// TIA Portal project "application-cp" (V18)

(* hardware
DEVICE "S7-1200 station_1"  S7-1200 Station
   slot 0: "Rack_0"  S7-1200 Rack  Rack  V1.0
   slot 1: "cpu"  CPU 1215C DC/DC/DC  6ES7 215-1AG40-0XB0  V4.6
*)

// ===== PLC "cpu"  CPU 1215C DC/DC/DC =====

VAR_GLOBAL   // PLC tag table "Default tag table"
   "Clock_Byte" AT %MB0 : Byte;
   "Clock_10Hz" AT %M0.0 : Bool;
   "Clock_5Hz" AT %M0.1 : Bool;
   "Clock_2.5Hz" AT %M0.2 : Bool;
   "Clock_2Hz" AT %M0.3 : Bool;
   "Clock_1.25Hz" AT %M0.4 : Bool;
   "Clock_1Hz" AT %M0.5 : Bool;
   "Clock_0.625Hz" AT %M0.6 : Bool;
   "Clock_0.5Hz" AT %M0.7 : Bool;
   "System_Byte" AT %MB1 : Byte;
   "FirstScan" AT %M1.0 : Bool;
   "DiagStatusUpdate" AT %M1.1 : Bool;
   "AlwaysTRUE" AT %M1.2 : Bool;
   "AlwaysFALSE" AT %M1.3 : Bool;
   "Tag_1" AT %M10.0 : Bool;
   "Tag_2" AT %M30.0 : Bool;
   "Tag_3" AT %M30.1 : Bool;
   "Tag_4" AT %M30.2 : Bool;
   "Tag_5" AT %M30.3 : Bool;
   "Tag_6" AT %M30.4 : Bool;
   "Tag_7" AT %M30.5 : Bool;
   "Tag_8" AT %M30.6 : Bool;
   "Tag_9" AT %M30.7 : Bool;
   "Tag_10" AT %M31.0 : Bool;
   "Tag_11" AT %M31.2 : Bool;
   "Tag_12" AT %M31.1 : Bool;
   "Tag_13" AT %M31.3 : Bool;
   "Tag_14" AT %M40.0 : Bool;
   "Tag_15" AT %M40.1 : Bool;
   "Tag_16" AT %M40.2 : Bool;
   "Tag_17" AT %M40.3 : Bool;
   "Tag_18" AT %M40.4 : Bool;
   "Tag_19" AT %M40.5 : Bool;
   "Tag_20" AT %M40.6 : Bool;
   "Tag_21" AT %M40.7 : Bool;
   "Tag_22" AT %M41.0 : Bool;
   "Tag_23" AT %M41.1 : Bool;
   "Tag_24" AT %M41.2 : Bool;
   "Tag_25" AT %M41.3 : Bool;
   "Tag_26" AT %M41.4 : Bool;
   "Tag_27" AT %M31.4 : Bool;
   "Tag_28" AT %M31.5 : Bool;
   "Tag_29" AT %M41.5 : Bool;
   "Tag_30" AT %M41.6 : Bool;
   "Tag_31" AT %M41.7 : Bool;
   "Tag_32" AT %M42.0 : Bool;
   "Tag_33" AT %M31.6 : Bool;
   "Tag_34" AT %M42.1 : Bool;
   "Tag_35" AT %M50.0 : Bool;
   "Tag_36" AT %M60.0 : Bool;
   "Tag_37" AT %M60.1 : Bool;
   "Tag_38" AT %M70.0 : Bool;
   "Tag_39" AT %M70.1 : Bool;
   "Tag_40" AT %M70.2 : Bool;
   "Tag_41" AT %M70.3 : Bool;
   "Tag_42" AT %M80.0 : Bool;
   "Tag_43" AT %M80.1 : Bool;
   "Tag_44" AT %M90.0 : Bool;
   "Tag_45" AT %M90.1 : Bool;
   "Tag_46" AT %M100.0 : Bool;
   "Tag_47" AT %M100.1 : Bool;
   "Tag_48" AT %M11.0 : Bool;
   "Tag_49" AT %M110.0 : Bool;
   "Tag_50" AT %M110.1 : Bool;
   "Tag_51" AT %M120.0 : Bool;
   "Tag_52" AT %M120.1 : Bool;
   "Tag_53" AT %M50.1 : Bool;
   "Tag_54" AT %M50.2 : Bool;
   "Tag_55" AT %M50.3 : Bool;
   "Tag_56" AT %M50.4 : Bool;
   "Tag_57" AT %M50.5 : Bool;
   "Tag_58" AT %M50.6 : Bool;
   "Tag_59" AT %M50.7 : Bool;
END_VAR

TYPE "Tank"
   STRUCT
      ID : Int;
      Sensor : Struct
         High : Bool;
         Low : Bool := true;
      END_STRUCT;
      Valve : Struct
         Drain : Bool;
         Source : Bool;
      END_STRUCT;
      Object : Struct
         Motor : Bool;
         Pump : Bool;
      END_STRUCT;
   END_STRUCT;
END_TYPE

TYPE "Line"
   STRUCT
      Supply : Struct
         Pump : Bool;
         Valve : Struct
            Caustic : Bool;
            Acid : Bool;
            Water : Bool;
            Rinse : Bool;
            Rice : Bool;
            Malt : Bool;
            Filter : Bool;
            Hops : Bool;
            Settling : Bool;
         END_STRUCT;
      END_STRUCT;
      "Return" : Struct
         Pump : Bool;
         Valve : Struct
            Caustic : Bool;
            Acid : Bool;
            Water : Bool;
            Rinse : Bool;
            Drain : Bool;
         END_STRUCT;
      END_STRUCT;
   END_STRUCT;
END_TYPE

DATA_BLOCK "DB_Tagforce"   // DB1
{ S7_Optimized_Access := 'FALSE' }
VERSION : 0.1
   VAR
      Button : Struct
         Run : Bool;
         Start : Bool;
         Mode : Bool;
         Clean : Struct
            Rice : Bool;
            Malt : Bool;
            Filter : Bool;
            Hops : Bool;
            Settling : Bool;
         END_STRUCT;
      END_STRUCT;
      Status : Struct
         Program : Struct
            Online : Bool;
            Offline : Bool;
            Idle : Bool;
            Busy : Bool;
         END_STRUCT;
         Mode : Struct
            Manual : Bool;
            Automatic : Bool;
         END_STRUCT;
         "Step" : Struct
            "1" : Bool;
            "2" : Bool;
            "3" : Bool;
            "4" : Bool;
            "5" : Bool;
            "6" : Bool;
            "7" : Bool;
         END_STRUCT;
         Clean : Struct
            Rice : Bool;
            Malt : Bool;
            Filter : Bool;
            Hops : Bool;
            Settling : Bool;
         END_STRUCT;
         Done : Bool;
      END_STRUCT;
      Lock : Struct
         Mode : Bool;
         "Step" : Struct
            "1" : Bool;
            "2" : Bool;
            "3" : Bool;
            "4" : Bool;
            "5" : Bool;
            "6" : Bool;
            "7" : Bool;
         END_STRUCT;
         Clean : Bool;
      END_STRUCT;
   END_VAR
BEGIN
END_DATA_BLOCK

DATA_BLOCK "DB_Tanks"   // DB2
{ S7_Optimized_Access := 'FALSE' }
VERSION : 0.1
   VAR
      Source : Struct
         Caustic : "Tank";
         Acid : "Tank";
         Water : "Tank";
         Rinse : "Tank";
      END_STRUCT;
      CIP : Struct
         Rice : "Tank";
         Malt : "Tank";
         Filter : "Tank";
         Hops : "Tank";
         Settling : "Tank";
         Current : "Tank";
         Backup : "Tank";
      END_STRUCT;
   END_VAR
BEGIN
   Source.Caustic.ID := 1;
   Source.Acid.ID := 2;
   Source.Water.ID := 3;
   Source.Rinse.ID := 4;
   CIP.Rice.ID := 5;
   CIP.Malt.ID := 6;
   CIP.Filter.ID := 7;
   CIP.Hops.ID := 8;
   CIP.Settling.ID := 9;
END_DATA_BLOCK

DATA_BLOCK "DB_Lines"   // DB3
{ S7_Optimized_Access := 'FALSE' }
VERSION : 0.1
   VAR
      Line : "Line";
   END_VAR
BEGIN
END_DATA_BLOCK

DATA_BLOCK "DB_Counter"   // DB37
{ S7_Optimized_Access := 'FALSE' }
VERSION : 0.1
   VAR
      Rice : Bool;
      Malt : Bool;
      Filter : Bool;
      Hops : Bool;
      Settling : Bool;
      Caustic : Bool;
      Acid : Bool;
      Water : Bool;
      Rinse : Bool;
      S7 : Bool;
      CC : Bool;
      CA : Bool;
      LM : Bool;
   END_VAR
BEGIN
END_DATA_BLOCK

// folder: System blocks/Program resources

DATA_BLOCK "IEC_Timer_0_DB"   // DB4
{ S7_Optimized_Access := 'TRUE' }
AUTHOR : Simatic
FAMILY : IEC
NAME : IEC_TMR
VERSION : 1.0
// stored: InstanceOfName IEC_TIMER
"IEC_TIMER"
BEGIN
END_DATA_BLOCK

DATA_BLOCK "IEC_Timer_0_DB_1"   // DB5
{ S7_Optimized_Access := 'TRUE' }
AUTHOR : Simatic
FAMILY : IEC
NAME : IEC_TMR
VERSION : 1.0
// stored: InstanceOfName IEC_TIMER
"IEC_TIMER"
BEGIN
END_DATA_BLOCK

DATA_BLOCK "IEC_Timer_0_DB_2"   // DB6
{ S7_Optimized_Access := 'TRUE' }
AUTHOR : Simatic
FAMILY : IEC
NAME : IEC_TMR
VERSION : 1.0
// stored: InstanceOfName IEC_TIMER
"IEC_TIMER"
BEGIN
END_DATA_BLOCK

DATA_BLOCK "IEC_Timer_0_DB_3"   // DB7
{ S7_Optimized_Access := 'TRUE' }
AUTHOR : Simatic
FAMILY : IEC
NAME : IEC_TMR
VERSION : 1.0
// stored: InstanceOfName IEC_TIMER
"IEC_TIMER"
BEGIN
END_DATA_BLOCK

DATA_BLOCK "IEC_Timer_0_DB_4"   // DB8
{ S7_Optimized_Access := 'TRUE' }
AUTHOR : Simatic
FAMILY : IEC
NAME : IEC_TMR
VERSION : 1.0
// stored: InstanceOfName IEC_TIMER
"IEC_TIMER"
BEGIN
END_DATA_BLOCK

DATA_BLOCK "IEC_Timer_0_DB_5"   // DB9
{ S7_Optimized_Access := 'TRUE' }
AUTHOR : Simatic
FAMILY : IEC
NAME : IEC_TMR
VERSION : 1.0
// stored: InstanceOfName IEC_TIMER
"IEC_TIMER"
BEGIN
END_DATA_BLOCK

DATA_BLOCK "IEC_Timer_0_DB_6"   // DB10
{ S7_Optimized_Access := 'TRUE' }
AUTHOR : Simatic
FAMILY : IEC
NAME : IEC_TMR
VERSION : 1.0
// stored: InstanceOfName IEC_TIMER
"IEC_TIMER"
BEGIN
END_DATA_BLOCK

DATA_BLOCK "IEC_Timer_0_DB_7"   // DB11
{ S7_Optimized_Access := 'TRUE' }
AUTHOR : Simatic
FAMILY : IEC
NAME : IEC_TMR
VERSION : 1.0
// stored: InstanceOfName IEC_TIMER
"IEC_TIMER"
BEGIN
END_DATA_BLOCK

DATA_BLOCK "IEC_Timer_0_DB_8"   // DB12
{ S7_Optimized_Access := 'TRUE' }
AUTHOR : Simatic
FAMILY : IEC
NAME : IEC_TMR
VERSION : 1.0
// stored: InstanceOfName IEC_TIMER
"IEC_TIMER"
BEGIN
END_DATA_BLOCK

DATA_BLOCK "IEC_Timer_0_DB_9"   // DB13
{ S7_Optimized_Access := 'TRUE' }
AUTHOR : Simatic
FAMILY : IEC
NAME : IEC_TMR
VERSION : 1.0
// stored: InstanceOfName IEC_TIMER
"IEC_TIMER"
BEGIN
END_DATA_BLOCK

DATA_BLOCK "IEC_Timer_0_DB_10"   // DB14
{ S7_Optimized_Access := 'TRUE' }
AUTHOR : Simatic
FAMILY : IEC
NAME : IEC_TMR
VERSION : 1.0
// stored: InstanceOfName IEC_TIMER
"IEC_TIMER"
BEGIN
END_DATA_BLOCK

DATA_BLOCK "IEC_Timer_0_DB_11"   // DB15
{ S7_Optimized_Access := 'TRUE' }
AUTHOR : Simatic
FAMILY : IEC
NAME : IEC_TMR
VERSION : 1.0
// stored: InstanceOfName IEC_TIMER
"IEC_TIMER"
BEGIN
END_DATA_BLOCK

DATA_BLOCK "IEC_Timer_0_DB_12"   // DB16
{ S7_Optimized_Access := 'TRUE' }
AUTHOR : Simatic
FAMILY : IEC
NAME : IEC_TMR
VERSION : 1.0
// stored: InstanceOfName IEC_TIMER
"IEC_TIMER"
BEGIN
END_DATA_BLOCK

DATA_BLOCK "IEC_Timer_0_DB_13"   // DB17
{ S7_Optimized_Access := 'TRUE' }
AUTHOR : Simatic
FAMILY : IEC
NAME : IEC_TMR
VERSION : 1.0
// stored: InstanceOfName IEC_TIMER
"IEC_TIMER"
BEGIN
END_DATA_BLOCK

DATA_BLOCK "IEC_Timer_0_DB_14"   // DB18
{ S7_Optimized_Access := 'TRUE' }
AUTHOR : Simatic
FAMILY : IEC
NAME : IEC_TMR
VERSION : 1.0
// stored: InstanceOfName IEC_TIMER
"IEC_TIMER"
BEGIN
END_DATA_BLOCK

DATA_BLOCK "IEC_Timer_0_DB_15"   // DB19
{ S7_Optimized_Access := 'TRUE' }
AUTHOR : Simatic
FAMILY : IEC
NAME : IEC_TMR
VERSION : 1.0
// stored: InstanceOfName IEC_TIMER
"IEC_TIMER"
BEGIN
END_DATA_BLOCK

DATA_BLOCK "IEC_Timer_0_DB_16"   // DB20
{ S7_Optimized_Access := 'TRUE' }
AUTHOR : Simatic
FAMILY : IEC
NAME : IEC_TMR
VERSION : 1.0
// stored: InstanceOfName IEC_TIMER
"IEC_TIMER"
BEGIN
END_DATA_BLOCK

DATA_BLOCK "IEC_Timer_0_DB_17"   // DB21
{ S7_Optimized_Access := 'TRUE' }
AUTHOR : Simatic
FAMILY : IEC
NAME : IEC_TMR
VERSION : 1.0
// stored: InstanceOfName IEC_TIMER
"IEC_TIMER"
BEGIN
END_DATA_BLOCK

DATA_BLOCK "IEC_Timer_0_DB_18"   // DB22
{ S7_Optimized_Access := 'TRUE' }
AUTHOR : Simatic
FAMILY : IEC
NAME : IEC_TMR
VERSION : 1.0
// stored: InstanceOfName IEC_TIMER
"IEC_TIMER"
BEGIN
END_DATA_BLOCK

DATA_BLOCK "IEC_Timer_0_DB_19"   // DB23
{ S7_Optimized_Access := 'TRUE' }
AUTHOR : Simatic
FAMILY : IEC
NAME : IEC_TMR
VERSION : 1.0
// stored: InstanceOfName IEC_TIMER
"IEC_TIMER"
BEGIN
END_DATA_BLOCK

DATA_BLOCK "IEC_Timer_0_DB_20"   // DB24
{ S7_Optimized_Access := 'TRUE' }
AUTHOR : Simatic
FAMILY : IEC
NAME : IEC_TMR
VERSION : 1.0
// stored: InstanceOfName IEC_TIMER
"IEC_TIMER"
BEGIN
END_DATA_BLOCK

DATA_BLOCK "IEC_Timer_0_DB_21"   // DB25
{ S7_Optimized_Access := 'TRUE' }
AUTHOR : Simatic
FAMILY : IEC
NAME : IEC_TMR
VERSION : 1.0
// stored: InstanceOfName IEC_TIMER
"IEC_TIMER"
BEGIN
END_DATA_BLOCK

DATA_BLOCK "IEC_Timer_0_DB_22"   // DB26
{ S7_Optimized_Access := 'TRUE' }
AUTHOR : Simatic
FAMILY : IEC
NAME : IEC_TMR
VERSION : 1.0
// stored: InstanceOfName IEC_TIMER
"IEC_TIMER"
BEGIN
END_DATA_BLOCK

DATA_BLOCK "IEC_Timer_0_DB_23"   // DB27
{ S7_Optimized_Access := 'TRUE' }
AUTHOR : Simatic
FAMILY : IEC
NAME : IEC_TMR
VERSION : 1.0
// stored: InstanceOfName IEC_TIMER
"IEC_TIMER"
BEGIN
END_DATA_BLOCK

DATA_BLOCK "IEC_Timer_0_DB_24"   // DB28
{ S7_Optimized_Access := 'TRUE' }
AUTHOR : Simatic
FAMILY : IEC
NAME : IEC_TMR
VERSION : 1.0
// stored: InstanceOfName IEC_TIMER
"IEC_TIMER"
BEGIN
END_DATA_BLOCK

DATA_BLOCK "IEC_Timer_0_DB_25"   // DB29
{ S7_Optimized_Access := 'TRUE' }
AUTHOR : Simatic
FAMILY : IEC
NAME : IEC_TMR
VERSION : 1.0
// stored: InstanceOfName IEC_TIMER
"IEC_TIMER"
BEGIN
END_DATA_BLOCK

DATA_BLOCK "IEC_Timer_0_DB_26"   // DB30
{ S7_Optimized_Access := 'TRUE' }
AUTHOR : Simatic
FAMILY : IEC
NAME : IEC_TMR
VERSION : 1.0
// stored: InstanceOfName IEC_TIMER
"IEC_TIMER"
BEGIN
END_DATA_BLOCK

DATA_BLOCK "IEC_Timer_0_DB_27"   // DB31
{ S7_Optimized_Access := 'TRUE' }
AUTHOR : Simatic
FAMILY : IEC
NAME : IEC_TMR
VERSION : 1.0
// stored: InstanceOfName IEC_TIMER
"IEC_TIMER"
BEGIN
END_DATA_BLOCK

DATA_BLOCK "IEC_Timer_0_DB_28"   // DB32
{ S7_Optimized_Access := 'TRUE' }
AUTHOR : Simatic
FAMILY : IEC
NAME : IEC_TMR
VERSION : 1.0
// stored: InstanceOfName IEC_TIMER
"IEC_TIMER"
BEGIN
END_DATA_BLOCK

DATA_BLOCK "IEC_Timer_0_DB_29"   // DB33
{ S7_Optimized_Access := 'TRUE' }
AUTHOR : Simatic
FAMILY : IEC
NAME : IEC_TMR
VERSION : 1.0
// stored: InstanceOfName IEC_TIMER
"IEC_TIMER"
BEGIN
END_DATA_BLOCK

DATA_BLOCK "IEC_Timer_0_DB_30"   // DB34
{ S7_Optimized_Access := 'TRUE' }
AUTHOR : Simatic
FAMILY : IEC
NAME : IEC_TMR
VERSION : 1.0
// stored: InstanceOfName IEC_TIMER
"IEC_TIMER"
BEGIN
END_DATA_BLOCK

// folder: (top level)

ORGANIZATION_BLOCK "Main"   // OB1, LAD, ProgramCycle
TITLE = "Main Program Sweep (Cycle)"
{ S7_Optimized_Access := 'TRUE' }
VERSION : 0.1
   VAR_INPUT
      Initial_Call : Bool;   // Initial call of this OB
      Remanence : Bool;   // =True, if remanent data are available
   END_VAR
   VAR_TEMP   // added for the SCL form of the ladder/FBD networks
      _w1 : Bool;
      _w2 : Bool;
      _w3 : Bool;
      _w4 : Bool;
      _w5 : Bool;
      _w6 : Bool;
      _w7 : Bool;
      _w8 : Bool;
      _w9 : Bool;
      _w10 : Bool;
      _w11 : Bool;
      _w12 : Bool;
      _w13 : Bool;
      _w14 : Bool;
      _w15 : Bool;
      _w16 : Bool;
   END_VAR
BEGIN

REGION Network 1: Program
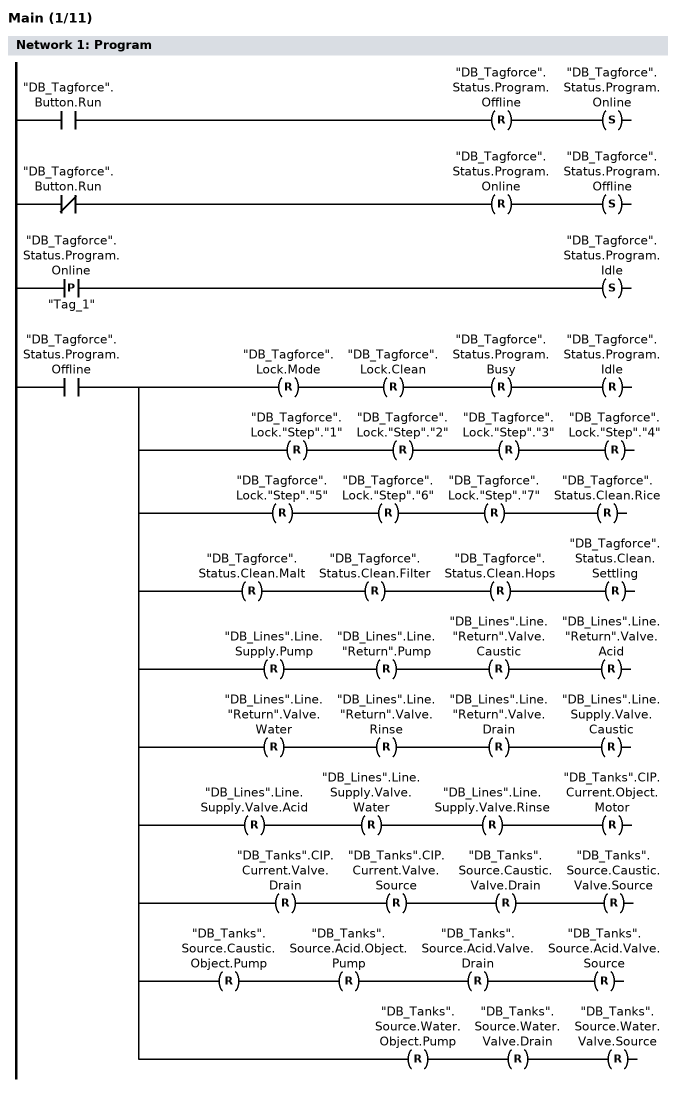
   RUNG wire#powerrail
      Contact( "DB_Tagforce".Button.Run )
      R_Coil( "DB_Tagforce".Status.Program.Offline )
      S_Coil( "DB_Tagforce".Status.Program.Online )
   END_RUNG
   RUNG wire#powerrail
      I_Contact( "DB_Tagforce".Button.Run )
      R_Coil( "DB_Tagforce".Status.Program.Online )
      S_Coil( "DB_Tagforce".Status.Program.Offline )
   END_RUNG
   RUNG wire#powerrail
      P_Contact(operand := "DB_Tagforce".Status.Program.Online, bit := "Tag_1")
      S_Coil( "DB_Tagforce".Status.Program.Idle )
   END_RUNG
   RUNG wire#powerrail
      Contact( "DB_Tagforce".Status.Program.Offline )
      wire#w1
      R_Coil( "DB_Tagforce".Lock.Mode )
      R_Coil( "DB_Tagforce".Lock.Clean )
      R_Coil( "DB_Tagforce".Status.Program.Busy )
      R_Coil( "DB_Tagforce".Status.Program.Idle )
   END_RUNG
   RUNG wire#w1
      R_Coil( "DB_Tagforce".Lock."Step"."1" )
      R_Coil( "DB_Tagforce".Lock."Step"."2" )
      R_Coil( "DB_Tagforce".Lock."Step"."3" )
      R_Coil( "DB_Tagforce".Lock."Step"."4" )
   END_RUNG
   RUNG wire#w1
      R_Coil( "DB_Tagforce".Lock."Step"."5" )
      R_Coil( "DB_Tagforce".Lock."Step"."6" )
      R_Coil( "DB_Tagforce".Lock."Step"."7" )
      R_Coil( "DB_Tagforce".Status.Clean.Rice )
   END_RUNG
   RUNG wire#w1
      R_Coil( "DB_Tagforce".Status.Clean.Malt )
      R_Coil( "DB_Tagforce".Status.Clean.Filter )
      R_Coil( "DB_Tagforce".Status.Clean.Hops )
      R_Coil( "DB_Tagforce".Status.Clean.Settling )
   END_RUNG
   RUNG wire#w1
      R_Coil( "DB_Lines".Line.Supply.Pump )
      R_Coil( "DB_Lines".Line."Return".Pump )
      R_Coil( "DB_Lines".Line."Return".Valve.Caustic )
      R_Coil( "DB_Lines".Line."Return".Valve.Acid )
   END_RUNG
   RUNG wire#w1
      R_Coil( "DB_Lines".Line."Return".Valve.Water )
      R_Coil( "DB_Lines".Line."Return".Valve.Rinse )
      R_Coil( "DB_Lines".Line."Return".Valve.Drain )
      R_Coil( "DB_Lines".Line.Supply.Valve.Caustic )
   END_RUNG
   RUNG wire#w1
      R_Coil( "DB_Lines".Line.Supply.Valve.Acid )
      R_Coil( "DB_Lines".Line.Supply.Valve.Water )
      R_Coil( "DB_Lines".Line.Supply.Valve.Rinse )
      R_Coil( "DB_Tanks".CIP.Current.Object.Motor )
   END_RUNG
   RUNG wire#w1
      R_Coil( "DB_Tanks".CIP.Current.Valve.Drain )
      R_Coil( "DB_Tanks".CIP.Current.Valve.Source )
      R_Coil( "DB_Tanks".Source.Caustic.Valve.Drain )
      R_Coil( "DB_Tanks".Source.Caustic.Valve.Source )
   END_RUNG
   RUNG wire#w1
      R_Coil( "DB_Tanks".Source.Caustic.Object.Pump )
      R_Coil( "DB_Tanks".Source.Acid.Object.Pump )
      R_Coil( "DB_Tanks".Source.Acid.Valve.Drain )
      R_Coil( "DB_Tanks".Source.Acid.Valve.Source )
   END_RUNG
   RUNG wire#w1
      R_Coil( "DB_Tanks".Source.Water.Object.Pump )
      R_Coil( "DB_Tanks".Source.Water.Valve.Drain )
      R_Coil( "DB_Tanks".Source.Water.Valve.Source )
   END_RUNG
   // the same network as SCL:
   IF "DB_Tagforce".Button.Run THEN
       "DB_Tagforce".Status.Program.Offline := FALSE;
       "DB_Tagforce".Status.Program.Online := TRUE;
   END_IF;
   IF NOT "DB_Tagforce".Button.Run THEN
       "DB_Tagforce".Status.Program.Online := FALSE;
       "DB_Tagforce".Status.Program.Offline := TRUE;
   END_IF;
   #_w1 := "DB_Tagforce".Status.Program.Online AND NOT "Tag_1";   // rising edge of "DB_Tagforce".Status.Program.Online
   "Tag_1" := "DB_Tagforce".Status.Program.Online;
   IF #_w1 THEN "DB_Tagforce".Status.Program.Idle := TRUE; END_IF;
   IF "DB_Tagforce".Status.Program.Offline THEN
       "DB_Tagforce".Lock.Mode := FALSE;
       "DB_Tagforce".Lock.Clean := FALSE;
       "DB_Tagforce".Status.Program.Busy := FALSE;
       "DB_Tagforce".Status.Program.Idle := FALSE;
       "DB_Tagforce".Lock."Step"."1" := FALSE;
       "DB_Tagforce".Lock."Step"."2" := FALSE;
       "DB_Tagforce".Lock."Step"."3" := FALSE;
       "DB_Tagforce".Lock."Step"."4" := FALSE;
       "DB_Tagforce".Lock."Step"."5" := FALSE;
       "DB_Tagforce".Lock."Step"."6" := FALSE;
       "DB_Tagforce".Lock."Step"."7" := FALSE;
       "DB_Tagforce".Status.Clean.Rice := FALSE;
       "DB_Tagforce".Status.Clean.Malt := FALSE;
       "DB_Tagforce".Status.Clean.Filter := FALSE;
       "DB_Tagforce".Status.Clean.Hops := FALSE;
       "DB_Tagforce".Status.Clean.Settling := FALSE;
       "DB_Lines".Line.Supply.Pump := FALSE;
       "DB_Lines".Line."Return".Pump := FALSE;
       "DB_Lines".Line."Return".Valve.Caustic := FALSE;
       "DB_Lines".Line."Return".Valve.Acid := FALSE;
       "DB_Lines".Line."Return".Valve.Water := FALSE;
       "DB_Lines".Line."Return".Valve.Rinse := FALSE;
       "DB_Lines".Line."Return".Valve.Drain := FALSE;
       "DB_Lines".Line.Supply.Valve.Caustic := FALSE;
       "DB_Lines".Line.Supply.Valve.Acid := FALSE;
       "DB_Lines".Line.Supply.Valve.Water := FALSE;
       "DB_Lines".Line.Supply.Valve.Rinse := FALSE;
       "DB_Tanks".CIP.Current.Object.Motor := FALSE;
       "DB_Tanks".CIP.Current.Valve.Drain := FALSE;
       "DB_Tanks".CIP.Current.Valve.Source := FALSE;
       "DB_Tanks".Source.Caustic.Valve.Drain := FALSE;
       "DB_Tanks".Source.Caustic.Valve.Source := FALSE;
       "DB_Tanks".Source.Caustic.Object.Pump := FALSE;
       "DB_Tanks".Source.Acid.Object.Pump := FALSE;
       "DB_Tanks".Source.Acid.Valve.Drain := FALSE;
       "DB_Tanks".Source.Acid.Valve.Source := FALSE;
       "DB_Tanks".Source.Water.Object.Pump := FALSE;
       "DB_Tanks".Source.Water.Valve.Drain := FALSE;
       "DB_Tanks".Source.Water.Valve.Source := FALSE;
   END_IF;
END_REGION

REGION Network 2: Mode
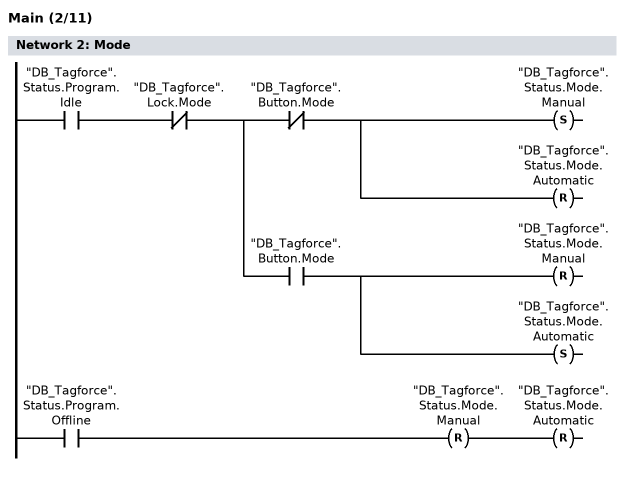
   RUNG wire#powerrail
      Contact( "DB_Tagforce".Status.Program.Idle )
      I_Contact( "DB_Tagforce".Lock.Mode )
      wire#w1
      I_Contact( "DB_Tagforce".Button.Mode )
      wire#w2
      S_Coil( "DB_Tagforce".Status.Mode.Manual )
   END_RUNG
   RUNG wire#w2
      R_Coil( "DB_Tagforce".Status.Mode.Automatic )
   END_RUNG
   RUNG wire#w1
      Contact( "DB_Tagforce".Button.Mode )
      wire#w3
      R_Coil( "DB_Tagforce".Status.Mode.Manual )
   END_RUNG
   RUNG wire#w3
      S_Coil( "DB_Tagforce".Status.Mode.Automatic )
   END_RUNG
   RUNG wire#powerrail
      Contact( "DB_Tagforce".Status.Program.Offline )
      R_Coil( "DB_Tagforce".Status.Mode.Manual )
      R_Coil( "DB_Tagforce".Status.Mode.Automatic )
   END_RUNG
   // the same network as SCL:
   #_w1 := "DB_Tagforce".Status.Program.Idle AND NOT "DB_Tagforce".Lock.Mode;
   IF #_w1 AND NOT "DB_Tagforce".Button.Mode THEN
       "DB_Tagforce".Status.Mode.Manual := TRUE;
       "DB_Tagforce".Status.Mode.Automatic := FALSE;
   END_IF;
   IF #_w1 AND "DB_Tagforce".Button.Mode THEN
       "DB_Tagforce".Status.Mode.Manual := FALSE;
       "DB_Tagforce".Status.Mode.Automatic := TRUE;
   END_IF;
   IF "DB_Tagforce".Status.Program.Offline THEN
       "DB_Tagforce".Status.Mode.Manual := FALSE;
       "DB_Tagforce".Status.Mode.Automatic := FALSE;
   END_IF;
END_REGION

REGION Network 3: Manual
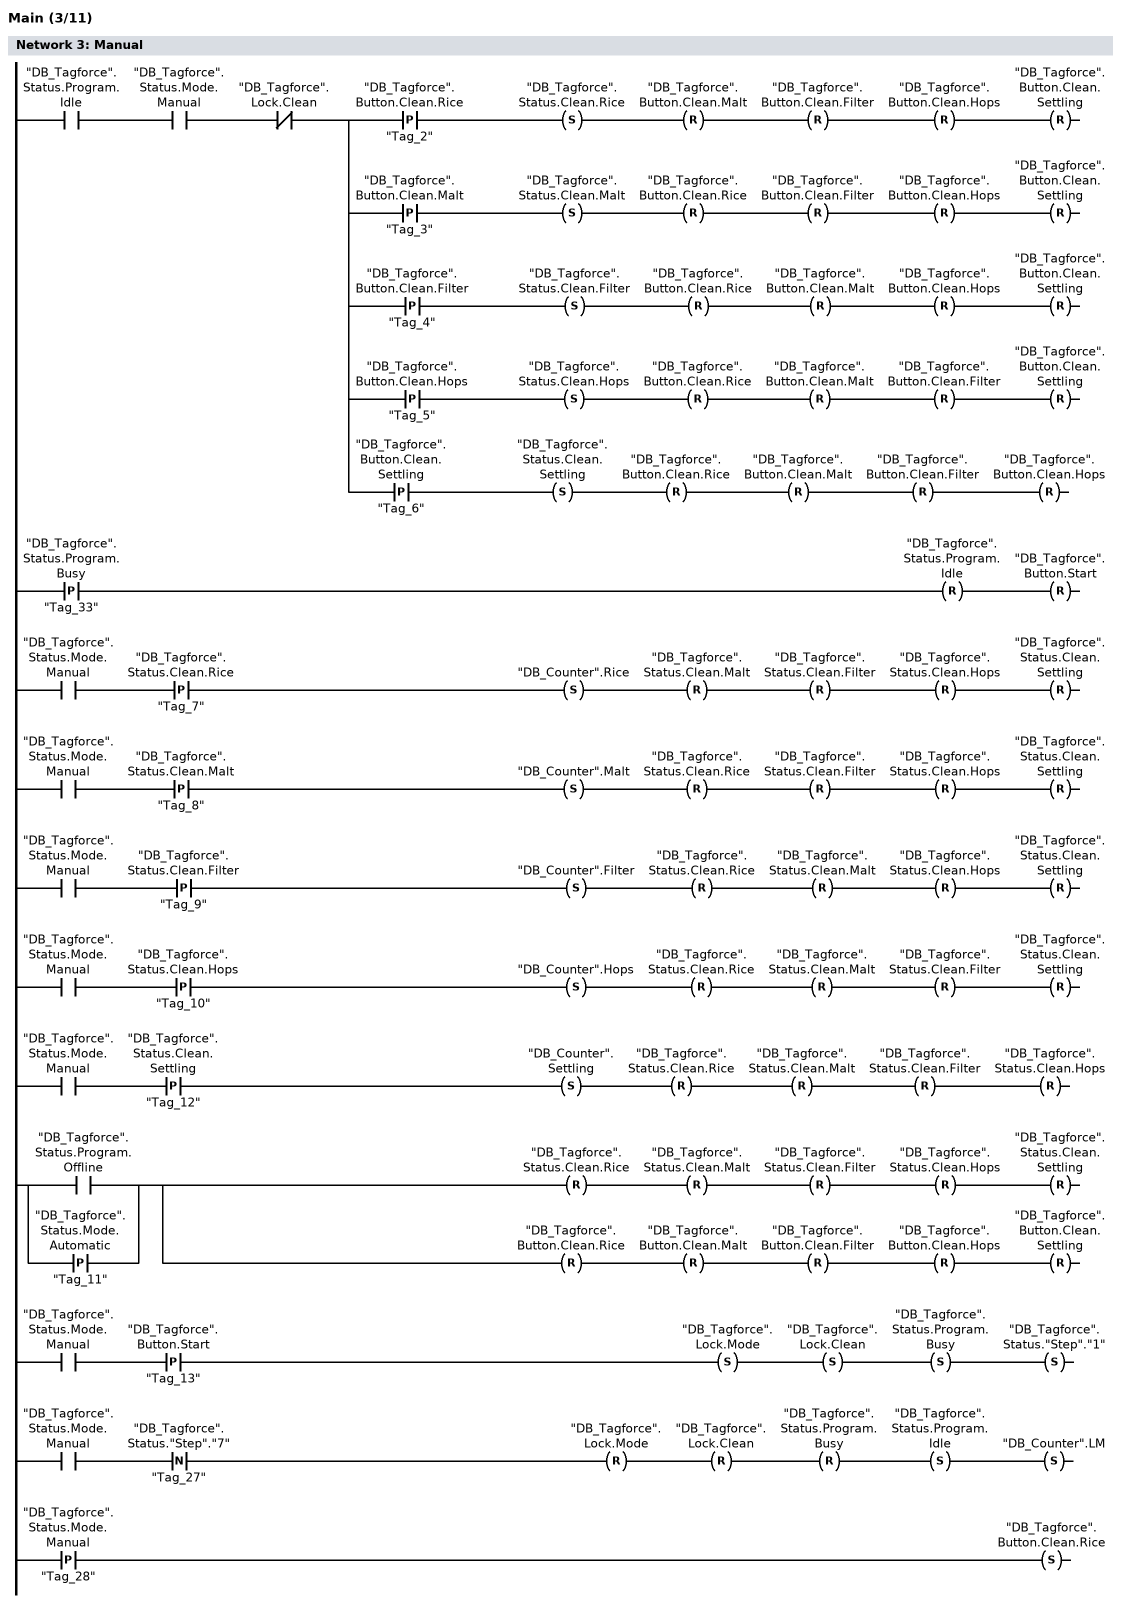
   RUNG wire#powerrail
      Contact( "DB_Tagforce".Status.Program.Idle )
      Contact( "DB_Tagforce".Status.Mode.Manual )
      I_Contact( "DB_Tagforce".Lock.Clean )
      wire#w1
      P_Contact(operand := "DB_Tagforce".Button.Clean.Rice, bit := "Tag_2")
      S_Coil( "DB_Tagforce".Status.Clean.Rice )
      R_Coil( "DB_Tagforce".Button.Clean.Malt )
      R_Coil( "DB_Tagforce".Button.Clean.Filter )
      R_Coil( "DB_Tagforce".Button.Clean.Hops )
      R_Coil( "DB_Tagforce".Button.Clean.Settling )
   END_RUNG
   RUNG wire#w1
      P_Contact(operand := "DB_Tagforce".Button.Clean.Malt, bit := "Tag_3")
      S_Coil( "DB_Tagforce".Status.Clean.Malt )
      R_Coil( "DB_Tagforce".Button.Clean.Rice )
      R_Coil( "DB_Tagforce".Button.Clean.Filter )
      R_Coil( "DB_Tagforce".Button.Clean.Hops )
      R_Coil( "DB_Tagforce".Button.Clean.Settling )
   END_RUNG
   RUNG wire#w1
      P_Contact(operand := "DB_Tagforce".Button.Clean.Filter, bit := "Tag_4")
      S_Coil( "DB_Tagforce".Status.Clean.Filter )
      R_Coil( "DB_Tagforce".Button.Clean.Rice )
      R_Coil( "DB_Tagforce".Button.Clean.Malt )
      R_Coil( "DB_Tagforce".Button.Clean.Hops )
      R_Coil( "DB_Tagforce".Button.Clean.Settling )
   END_RUNG
   RUNG wire#w1
      P_Contact(operand := "DB_Tagforce".Button.Clean.Hops, bit := "Tag_5")
      S_Coil( "DB_Tagforce".Status.Clean.Hops )
      R_Coil( "DB_Tagforce".Button.Clean.Rice )
      R_Coil( "DB_Tagforce".Button.Clean.Malt )
      R_Coil( "DB_Tagforce".Button.Clean.Filter )
      R_Coil( "DB_Tagforce".Button.Clean.Settling )
   END_RUNG
   RUNG wire#w1
      P_Contact(operand := "DB_Tagforce".Button.Clean.Settling, bit := "Tag_6")
      S_Coil( "DB_Tagforce".Status.Clean.Settling )
      R_Coil( "DB_Tagforce".Button.Clean.Rice )
      R_Coil( "DB_Tagforce".Button.Clean.Malt )
      R_Coil( "DB_Tagforce".Button.Clean.Filter )
      R_Coil( "DB_Tagforce".Button.Clean.Hops )
   END_RUNG
   RUNG wire#powerrail
      P_Contact(operand := "DB_Tagforce".Status.Program.Busy, bit := "Tag_33")
      R_Coil( "DB_Tagforce".Status.Program.Idle )
      R_Coil( "DB_Tagforce".Button.Start )
   END_RUNG
   RUNG wire#powerrail
      Contact( "DB_Tagforce".Status.Mode.Manual )
      P_Contact(operand := "DB_Tagforce".Status.Clean.Rice, bit := "Tag_7")
      S_Coil( "DB_Counter".Rice )
      R_Coil( "DB_Tagforce".Status.Clean.Malt )
      R_Coil( "DB_Tagforce".Status.Clean.Filter )
      R_Coil( "DB_Tagforce".Status.Clean.Hops )
      R_Coil( "DB_Tagforce".Status.Clean.Settling )
   END_RUNG
   RUNG wire#powerrail
      Contact( "DB_Tagforce".Status.Mode.Manual )
      P_Contact(operand := "DB_Tagforce".Status.Clean.Malt, bit := "Tag_8")
      S_Coil( "DB_Counter".Malt )
      R_Coil( "DB_Tagforce".Status.Clean.Rice )
      R_Coil( "DB_Tagforce".Status.Clean.Filter )
      R_Coil( "DB_Tagforce".Status.Clean.Hops )
      R_Coil( "DB_Tagforce".Status.Clean.Settling )
   END_RUNG
   RUNG wire#powerrail
      Contact( "DB_Tagforce".Status.Mode.Manual )
      P_Contact(operand := "DB_Tagforce".Status.Clean.Filter, bit := "Tag_9")
      S_Coil( "DB_Counter".Filter )
      R_Coil( "DB_Tagforce".Status.Clean.Rice )
      R_Coil( "DB_Tagforce".Status.Clean.Malt )
      R_Coil( "DB_Tagforce".Status.Clean.Hops )
      R_Coil( "DB_Tagforce".Status.Clean.Settling )
   END_RUNG
   RUNG wire#powerrail
      Contact( "DB_Tagforce".Status.Mode.Manual )
      P_Contact(operand := "DB_Tagforce".Status.Clean.Hops, bit := "Tag_10")
      S_Coil( "DB_Counter".Hops )
      R_Coil( "DB_Tagforce".Status.Clean.Rice )
      R_Coil( "DB_Tagforce".Status.Clean.Malt )
      R_Coil( "DB_Tagforce".Status.Clean.Filter )
      R_Coil( "DB_Tagforce".Status.Clean.Settling )
   END_RUNG
   RUNG wire#powerrail
      Contact( "DB_Tagforce".Status.Mode.Manual )
      P_Contact(operand := "DB_Tagforce".Status.Clean.Settling, bit := "Tag_12")
      S_Coil( "DB_Counter".Settling )
      R_Coil( "DB_Tagforce".Status.Clean.Rice )
      R_Coil( "DB_Tagforce".Status.Clean.Malt )
      R_Coil( "DB_Tagforce".Status.Clean.Filter )
      R_Coil( "DB_Tagforce".Status.Clean.Hops )
   END_RUNG
   RUNG wire#powerrail
      Contact( "DB_Tagforce".Status.Program.Offline )
      wire#w2
      R_Coil( "DB_Tagforce".Status.Clean.Rice )
      R_Coil( "DB_Tagforce".Status.Clean.Malt )
      R_Coil( "DB_Tagforce".Status.Clean.Filter )
      R_Coil( "DB_Tagforce".Status.Clean.Hops )
      R_Coil( "DB_Tagforce".Status.Clean.Settling )
   END_RUNG
   RUNG wire#powerrail
      P_Contact(operand := "DB_Tagforce".Status.Mode.Automatic, bit := "Tag_11")
   END_RUNG wire#w2
   RUNG wire#w2
      R_Coil( "DB_Tagforce".Button.Clean.Rice )
      R_Coil( "DB_Tagforce".Button.Clean.Malt )
      R_Coil( "DB_Tagforce".Button.Clean.Filter )
      R_Coil( "DB_Tagforce".Button.Clean.Hops )
      R_Coil( "DB_Tagforce".Button.Clean.Settling )
   END_RUNG
   RUNG wire#powerrail
      Contact( "DB_Tagforce".Status.Mode.Manual )
      P_Contact(operand := "DB_Tagforce".Button.Start, bit := "Tag_13")
      S_Coil( "DB_Tagforce".Lock.Mode )
      S_Coil( "DB_Tagforce".Lock.Clean )
      S_Coil( "DB_Tagforce".Status.Program.Busy )
      S_Coil( "DB_Tagforce".Status."Step"."1" )
   END_RUNG
   RUNG wire#powerrail
      Contact( "DB_Tagforce".Status.Mode.Manual )
      N_Contact(operand := "DB_Tagforce".Status."Step"."7", bit := "Tag_27")
      R_Coil( "DB_Tagforce".Lock.Mode )
      R_Coil( "DB_Tagforce".Lock.Clean )
      R_Coil( "DB_Tagforce".Status.Program.Busy )
      S_Coil( "DB_Tagforce".Status.Program.Idle )
      S_Coil( "DB_Counter".LM )
   END_RUNG
   RUNG wire#powerrail
      P_Contact(operand := "DB_Tagforce".Status.Mode.Manual, bit := "Tag_28")
      S_Coil( "DB_Tagforce".Button.Clean.Rice )
   END_RUNG
   // the same network as SCL:
   #_w1 := "DB_Tagforce".Status.Program.Idle AND "DB_Tagforce".Status.Mode.Manual AND NOT "DB_Tagforce".Lock.Clean;
   #_w2 := #_w1 AND "DB_Tagforce".Button.Clean.Rice AND NOT "Tag_2";   // rising edge of "DB_Tagforce".Button.Clean.Rice
   "Tag_2" := "DB_Tagforce".Button.Clean.Rice;
   IF #_w2 THEN
       "DB_Tagforce".Status.Clean.Rice := TRUE;
       "DB_Tagforce".Button.Clean.Malt := FALSE;
       "DB_Tagforce".Button.Clean.Filter := FALSE;
       "DB_Tagforce".Button.Clean.Hops := FALSE;
       "DB_Tagforce".Button.Clean.Settling := FALSE;
   END_IF;
   #_w3 := #_w1 AND "DB_Tagforce".Button.Clean.Malt AND NOT "Tag_3";   // rising edge of "DB_Tagforce".Button.Clean.Malt
   "Tag_3" := "DB_Tagforce".Button.Clean.Malt;
   IF #_w3 THEN
       "DB_Tagforce".Status.Clean.Malt := TRUE;
       "DB_Tagforce".Button.Clean.Rice := FALSE;
       "DB_Tagforce".Button.Clean.Filter := FALSE;
       "DB_Tagforce".Button.Clean.Hops := FALSE;
       "DB_Tagforce".Button.Clean.Settling := FALSE;
   END_IF;
   #_w4 := #_w1 AND "DB_Tagforce".Button.Clean.Filter AND NOT "Tag_4";   // rising edge of "DB_Tagforce".Button.Clean.Filter
   "Tag_4" := "DB_Tagforce".Button.Clean.Filter;
   IF #_w4 THEN
       "DB_Tagforce".Status.Clean.Filter := TRUE;
       "DB_Tagforce".Button.Clean.Rice := FALSE;
       "DB_Tagforce".Button.Clean.Malt := FALSE;
       "DB_Tagforce".Button.Clean.Hops := FALSE;
       "DB_Tagforce".Button.Clean.Settling := FALSE;
   END_IF;
   #_w5 := #_w1 AND "DB_Tagforce".Button.Clean.Hops AND NOT "Tag_5";   // rising edge of "DB_Tagforce".Button.Clean.Hops
   "Tag_5" := "DB_Tagforce".Button.Clean.Hops;
   IF #_w5 THEN
       "DB_Tagforce".Status.Clean.Hops := TRUE;
       "DB_Tagforce".Button.Clean.Rice := FALSE;
       "DB_Tagforce".Button.Clean.Malt := FALSE;
       "DB_Tagforce".Button.Clean.Filter := FALSE;
       "DB_Tagforce".Button.Clean.Settling := FALSE;
   END_IF;
   #_w6 := #_w1 AND "DB_Tagforce".Button.Clean.Settling AND NOT "Tag_6";   // rising edge of "DB_Tagforce".Button.Clean.Settling
   "Tag_6" := "DB_Tagforce".Button.Clean.Settling;
   IF #_w6 THEN
       "DB_Tagforce".Status.Clean.Settling := TRUE;
       "DB_Tagforce".Button.Clean.Rice := FALSE;
       "DB_Tagforce".Button.Clean.Malt := FALSE;
       "DB_Tagforce".Button.Clean.Filter := FALSE;
       "DB_Tagforce".Button.Clean.Hops := FALSE;
   END_IF;
   #_w7 := "DB_Tagforce".Status.Program.Busy AND NOT "Tag_33";   // rising edge of "DB_Tagforce".Status.Program.Busy
   "Tag_33" := "DB_Tagforce".Status.Program.Busy;
   IF #_w7 THEN
       "DB_Tagforce".Status.Program.Idle := FALSE;
       "DB_Tagforce".Button.Start := FALSE;
   END_IF;
   #_w8 := "DB_Tagforce".Status.Mode.Manual AND "DB_Tagforce".Status.Clean.Rice AND NOT "Tag_7";   // rising edge of "DB_Tagforce".Status.Clean.Rice
   "Tag_7" := "DB_Tagforce".Status.Clean.Rice;
   IF #_w8 THEN
       "DB_Counter".Rice := TRUE;
       "DB_Tagforce".Status.Clean.Malt := FALSE;
       "DB_Tagforce".Status.Clean.Filter := FALSE;
       "DB_Tagforce".Status.Clean.Hops := FALSE;
       "DB_Tagforce".Status.Clean.Settling := FALSE;
   END_IF;
   #_w9 := "DB_Tagforce".Status.Mode.Manual AND "DB_Tagforce".Status.Clean.Malt AND NOT "Tag_8";   // rising edge of "DB_Tagforce".Status.Clean.Malt
   "Tag_8" := "DB_Tagforce".Status.Clean.Malt;
   IF #_w9 THEN
       "DB_Counter".Malt := TRUE;
       "DB_Tagforce".Status.Clean.Rice := FALSE;
       "DB_Tagforce".Status.Clean.Filter := FALSE;
       "DB_Tagforce".Status.Clean.Hops := FALSE;
       "DB_Tagforce".Status.Clean.Settling := FALSE;
   END_IF;
   #_w10 := "DB_Tagforce".Status.Mode.Manual AND "DB_Tagforce".Status.Clean.Filter AND NOT "Tag_9";   // rising edge of "DB_Tagforce".Status.Clean.Filter
   "Tag_9" := "DB_Tagforce".Status.Clean.Filter;
   IF #_w10 THEN
       "DB_Counter".Filter := TRUE;
       "DB_Tagforce".Status.Clean.Rice := FALSE;
       "DB_Tagforce".Status.Clean.Malt := FALSE;
       "DB_Tagforce".Status.Clean.Hops := FALSE;
       "DB_Tagforce".Status.Clean.Settling := FALSE;
   END_IF;
   #_w11 := "DB_Tagforce".Status.Mode.Manual AND "DB_Tagforce".Status.Clean.Hops AND NOT "Tag_10";   // rising edge of "DB_Tagforce".Status.Clean.Hops
   "Tag_10" := "DB_Tagforce".Status.Clean.Hops;
   IF #_w11 THEN
       "DB_Counter".Hops := TRUE;
       "DB_Tagforce".Status.Clean.Rice := FALSE;
       "DB_Tagforce".Status.Clean.Malt := FALSE;
       "DB_Tagforce".Status.Clean.Filter := FALSE;
       "DB_Tagforce".Status.Clean.Settling := FALSE;
   END_IF;
   #_w12 := "DB_Tagforce".Status.Mode.Manual AND "DB_Tagforce".Status.Clean.Settling AND NOT "Tag_12";   // rising edge of "DB_Tagforce".Status.Clean.Settling
   "Tag_12" := "DB_Tagforce".Status.Clean.Settling;
   IF #_w12 THEN
       "DB_Counter".Settling := TRUE;
       "DB_Tagforce".Status.Clean.Rice := FALSE;
       "DB_Tagforce".Status.Clean.Malt := FALSE;
       "DB_Tagforce".Status.Clean.Filter := FALSE;
       "DB_Tagforce".Status.Clean.Hops := FALSE;
   END_IF;
   #_w13 := "DB_Tagforce".Status.Mode.Automatic AND NOT "Tag_11";   // rising edge of "DB_Tagforce".Status.Mode.Automatic
   "Tag_11" := "DB_Tagforce".Status.Mode.Automatic;
   IF "DB_Tagforce".Status.Program.Offline OR #_w13 THEN
       "DB_Tagforce".Status.Clean.Rice := FALSE;
       "DB_Tagforce".Status.Clean.Malt := FALSE;
       "DB_Tagforce".Status.Clean.Filter := FALSE;
       "DB_Tagforce".Status.Clean.Hops := FALSE;
       "DB_Tagforce".Status.Clean.Settling := FALSE;
       "DB_Tagforce".Button.Clean.Rice := FALSE;
       "DB_Tagforce".Button.Clean.Malt := FALSE;
       "DB_Tagforce".Button.Clean.Filter := FALSE;
       "DB_Tagforce".Button.Clean.Hops := FALSE;
       "DB_Tagforce".Button.Clean.Settling := FALSE;
   END_IF;
   #_w14 := "DB_Tagforce".Status.Mode.Manual AND "DB_Tagforce".Button.Start AND NOT "Tag_13";   // rising edge of "DB_Tagforce".Button.Start
   "Tag_13" := "DB_Tagforce".Button.Start;
   IF #_w14 THEN
       "DB_Tagforce".Lock.Mode := TRUE;
       "DB_Tagforce".Lock.Clean := TRUE;
       "DB_Tagforce".Status.Program.Busy := TRUE;
       "DB_Tagforce".Status."Step"."1" := TRUE;
   END_IF;
   #_w15 := "DB_Tagforce".Status.Mode.Manual AND NOT "DB_Tagforce".Status."Step"."7" AND "Tag_27";   // falling edge of "DB_Tagforce".Status."Step"."7"
   "Tag_27" := "DB_Tagforce".Status."Step"."7";
   IF #_w15 THEN
       "DB_Tagforce".Lock.Mode := FALSE;
       "DB_Tagforce".Lock.Clean := FALSE;
       "DB_Tagforce".Status.Program.Busy := FALSE;
       "DB_Tagforce".Status.Program.Idle := TRUE;
       "DB_Counter".LM := TRUE;
   END_IF;
   #_w16 := "DB_Tagforce".Status.Mode.Manual AND NOT "Tag_28";   // rising edge of "DB_Tagforce".Status.Mode.Manual
   "Tag_28" := "DB_Tagforce".Status.Mode.Manual;
   IF #_w16 THEN "DB_Tagforce".Button.Clean.Rice := TRUE; END_IF;
END_REGION

REGION Network 4: Automatic
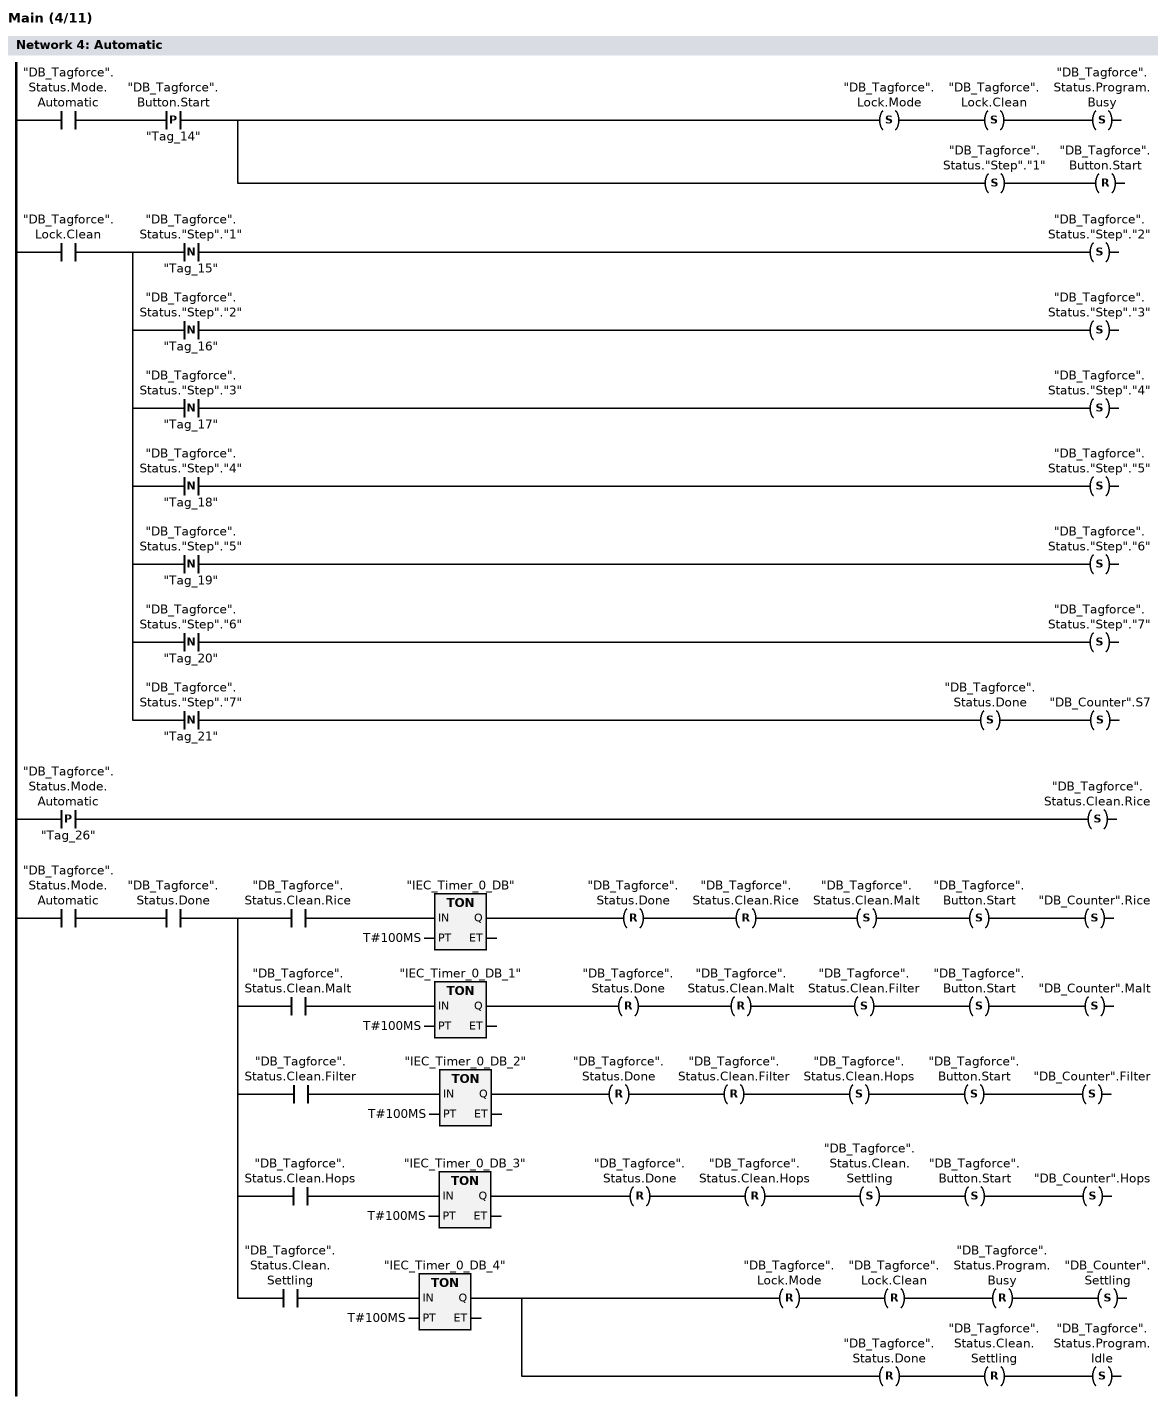
   #_w1 := "DB_Tagforce".Status.Mode.Automatic AND "DB_Tagforce".Button.Start AND NOT "Tag_14";   // rising edge of "DB_Tagforce".Button.Start
   "Tag_14" := "DB_Tagforce".Button.Start;
   IF #_w1 THEN
       "DB_Tagforce".Lock.Mode := TRUE;
       "DB_Tagforce".Lock.Clean := TRUE;
       "DB_Tagforce".Status.Program.Busy := TRUE;
       "DB_Tagforce".Status."Step"."1" := TRUE;
       "DB_Tagforce".Button.Start := FALSE;
   END_IF;
   #_w2 := "DB_Tagforce".Lock.Clean AND NOT "DB_Tagforce".Status."Step"."1" AND "Tag_15";   // falling edge of "DB_Tagforce".Status."Step"."1"
   "Tag_15" := "DB_Tagforce".Status."Step"."1";
   IF #_w2 THEN "DB_Tagforce".Status."Step"."2" := TRUE; END_IF;
   #_w3 := "DB_Tagforce".Lock.Clean AND NOT "DB_Tagforce".Status."Step"."2" AND "Tag_16";   // falling edge of "DB_Tagforce".Status."Step"."2"
   "Tag_16" := "DB_Tagforce".Status."Step"."2";
   IF #_w3 THEN "DB_Tagforce".Status."Step"."3" := TRUE; END_IF;
   #_w4 := "DB_Tagforce".Lock.Clean AND NOT "DB_Tagforce".Status."Step"."3" AND "Tag_17";   // falling edge of "DB_Tagforce".Status."Step"."3"
   "Tag_17" := "DB_Tagforce".Status."Step"."3";
   IF #_w4 THEN "DB_Tagforce".Status."Step"."4" := TRUE; END_IF;
   #_w5 := "DB_Tagforce".Lock.Clean AND NOT "DB_Tagforce".Status."Step"."4" AND "Tag_18";   // falling edge of "DB_Tagforce".Status."Step"."4"
   "Tag_18" := "DB_Tagforce".Status."Step"."4";
   IF #_w5 THEN "DB_Tagforce".Status."Step"."5" := TRUE; END_IF;
   #_w6 := "DB_Tagforce".Lock.Clean AND NOT "DB_Tagforce".Status."Step"."5" AND "Tag_19";   // falling edge of "DB_Tagforce".Status."Step"."5"
   "Tag_19" := "DB_Tagforce".Status."Step"."5";
   IF #_w6 THEN "DB_Tagforce".Status."Step"."6" := TRUE; END_IF;
   #_w7 := "DB_Tagforce".Lock.Clean AND NOT "DB_Tagforce".Status."Step"."6" AND "Tag_20";   // falling edge of "DB_Tagforce".Status."Step"."6"
   "Tag_20" := "DB_Tagforce".Status."Step"."6";
   IF #_w7 THEN "DB_Tagforce".Status."Step"."7" := TRUE; END_IF;
   #_w8 := "DB_Tagforce".Lock.Clean AND NOT "DB_Tagforce".Status."Step"."7" AND "Tag_21";   // falling edge of "DB_Tagforce".Status."Step"."7"
   "Tag_21" := "DB_Tagforce".Status."Step"."7";
   IF #_w8 THEN
       "DB_Tagforce".Status.Done := TRUE;
       "DB_Counter".S7 := TRUE;
   END_IF;
   #_w9 := "DB_Tagforce".Status.Mode.Automatic AND NOT "Tag_26";   // rising edge of "DB_Tagforce".Status.Mode.Automatic
   "Tag_26" := "DB_Tagforce".Status.Mode.Automatic;
   IF #_w9 THEN "DB_Tagforce".Status.Clean.Rice := TRUE; END_IF;
   #_w10 := "DB_Tagforce".Status.Mode.Automatic AND "DB_Tagforce".Status.Done;
   "IEC_Timer_0_DB".TON(IN := #_w10 AND "DB_Tagforce".Status.Clean.Rice, PT := T#100MS);
   IF "IEC_Timer_0_DB".Q THEN
       "DB_Tagforce".Status.Done := FALSE;
       "DB_Tagforce".Status.Clean.Rice := FALSE;
       "DB_Tagforce".Status.Clean.Malt := TRUE;
       "DB_Tagforce".Button.Start := TRUE;
       "DB_Counter".Rice := TRUE;
   END_IF;
   "IEC_Timer_0_DB_1".TON(IN := #_w10 AND "DB_Tagforce".Status.Clean.Malt, PT := T#100MS);
   IF "IEC_Timer_0_DB_1".Q THEN
       "DB_Tagforce".Status.Done := FALSE;
       "DB_Tagforce".Status.Clean.Malt := FALSE;
       "DB_Tagforce".Status.Clean.Filter := TRUE;
       "DB_Tagforce".Button.Start := TRUE;
       "DB_Counter".Malt := TRUE;
   END_IF;
   "IEC_Timer_0_DB_2".TON(IN := #_w10 AND "DB_Tagforce".Status.Clean.Filter, PT := T#100MS);
   IF "IEC_Timer_0_DB_2".Q THEN
       "DB_Tagforce".Status.Done := FALSE;
       "DB_Tagforce".Status.Clean.Filter := FALSE;
       "DB_Tagforce".Status.Clean.Hops := TRUE;
       "DB_Tagforce".Button.Start := TRUE;
       "DB_Counter".Filter := TRUE;
   END_IF;
   "IEC_Timer_0_DB_3".TON(IN := #_w10 AND "DB_Tagforce".Status.Clean.Hops, PT := T#100MS);
   IF "IEC_Timer_0_DB_3".Q THEN
       "DB_Tagforce".Status.Done := FALSE;
       "DB_Tagforce".Status.Clean.Hops := FALSE;
       "DB_Tagforce".Status.Clean.Settling := TRUE;
       "DB_Tagforce".Button.Start := TRUE;
       "DB_Counter".Hops := TRUE;
   END_IF;
   "IEC_Timer_0_DB_4".TON(IN := #_w10 AND "DB_Tagforce".Status.Clean.Settling, PT := T#100MS);
   IF "IEC_Timer_0_DB_4".Q THEN
       "DB_Tagforce".Lock.Mode := FALSE;
       "DB_Tagforce".Lock.Clean := FALSE;
       "DB_Tagforce".Status.Program.Busy := FALSE;
       "DB_Counter".Settling := TRUE;
       "DB_Tagforce".Status.Done := FALSE;
       "DB_Tagforce".Status.Clean.Settling := FALSE;
       "DB_Tagforce".Status.Program.Idle := TRUE;
   END_IF;
END_REGION

REGION Network 5: Step 1: Pre Empty
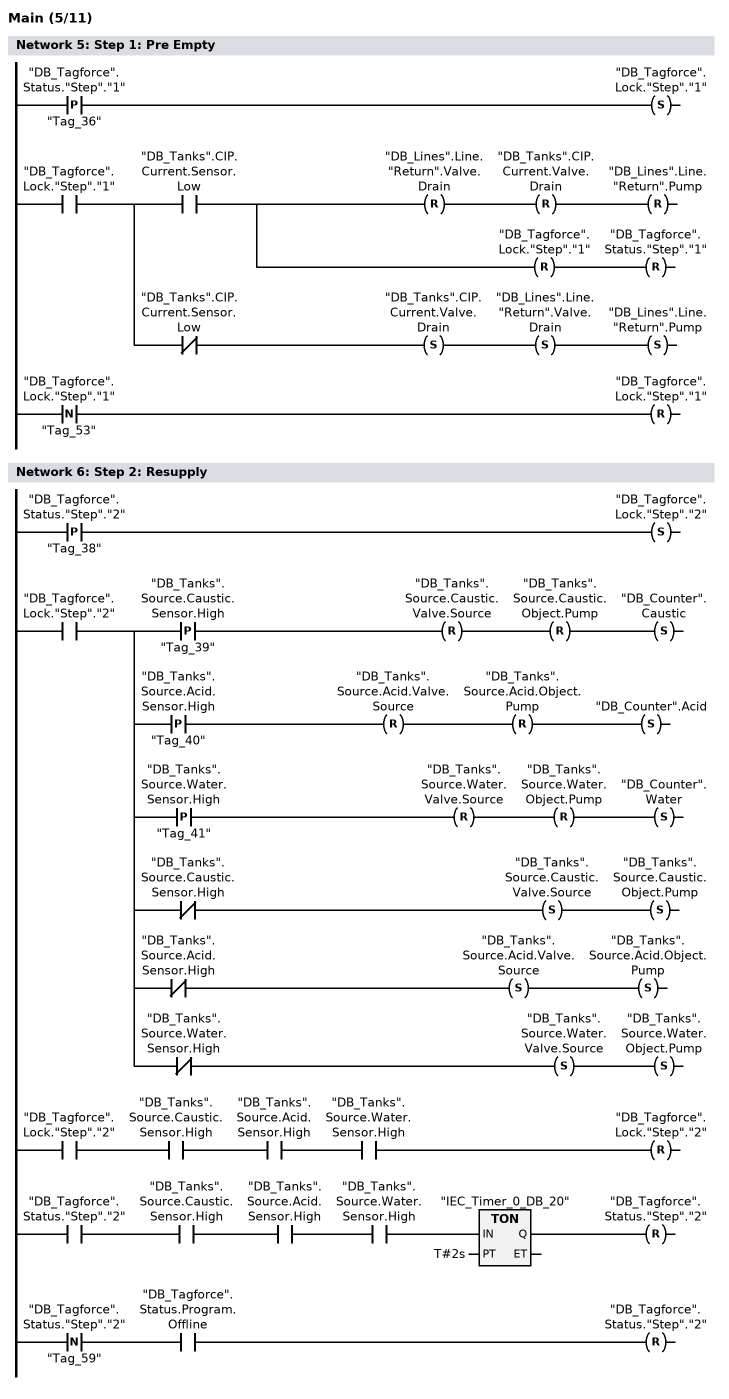
   RUNG wire#powerrail
      P_Contact(operand := "DB_Tagforce".Status."Step"."1", bit := "Tag_36")
      S_Coil( "DB_Tagforce".Lock."Step"."1" )
   END_RUNG
   RUNG wire#powerrail
      Contact( "DB_Tagforce".Lock."Step"."1" )
      wire#w1
      Contact( "DB_Tanks".CIP.Current.Sensor.Low )
      wire#w2
      R_Coil( "DB_Lines".Line."Return".Valve.Drain )
      R_Coil( "DB_Tanks".CIP.Current.Valve.Drain )
      R_Coil( "DB_Lines".Line."Return".Pump )
   END_RUNG
   RUNG wire#w2
      R_Coil( "DB_Tagforce".Lock."Step"."1" )
      R_Coil( "DB_Tagforce".Status."Step"."1" )
   END_RUNG
   RUNG wire#w1
      I_Contact( "DB_Tanks".CIP.Current.Sensor.Low )
      S_Coil( "DB_Tanks".CIP.Current.Valve.Drain )
      S_Coil( "DB_Lines".Line."Return".Valve.Drain )
      S_Coil( "DB_Lines".Line."Return".Pump )
   END_RUNG
   RUNG wire#powerrail
      N_Contact(operand := "DB_Tagforce".Lock."Step"."1", bit := "Tag_53")
      R_Coil( "DB_Tagforce".Lock."Step"."1" )
   END_RUNG
   // the same network as SCL:
   #_w1 := "DB_Tagforce".Status."Step"."1" AND NOT "Tag_36";   // rising edge of "DB_Tagforce".Status."Step"."1"
   "Tag_36" := "DB_Tagforce".Status."Step"."1";
   IF #_w1 THEN "DB_Tagforce".Lock."Step"."1" := TRUE; END_IF;
   IF "DB_Tagforce".Lock."Step"."1" AND "DB_Tanks".CIP.Current.Sensor.Low THEN
       "DB_Lines".Line."Return".Valve.Drain := FALSE;
       "DB_Tanks".CIP.Current.Valve.Drain := FALSE;
       "DB_Lines".Line."Return".Pump := FALSE;
   END_IF;
   #_w2 := "DB_Tagforce".Lock."Step"."1" AND "DB_Tanks".CIP.Current.Sensor.Low;
   #_w3 := "DB_Tagforce".Lock."Step"."1";
   IF #_w2 THEN
       "DB_Tagforce".Lock."Step"."1" := FALSE;
       "DB_Tagforce".Status."Step"."1" := FALSE;
   END_IF;
   IF #_w3 AND NOT "DB_Tanks".CIP.Current.Sensor.Low THEN
       "DB_Tanks".CIP.Current.Valve.Drain := TRUE;
       "DB_Lines".Line."Return".Valve.Drain := TRUE;
       "DB_Lines".Line."Return".Pump := TRUE;
   END_IF;
   #_w4 := NOT "DB_Tagforce".Lock."Step"."1" AND "Tag_53";   // falling edge of "DB_Tagforce".Lock."Step"."1"
   "Tag_53" := "DB_Tagforce".Lock."Step"."1";
   IF #_w4 THEN "DB_Tagforce".Lock."Step"."1" := FALSE; END_IF;
END_REGION

REGION Network 6: Step 2: Resupply
   #_w1 := "DB_Tagforce".Status."Step"."2" AND NOT "Tag_38";   // rising edge of "DB_Tagforce".Status."Step"."2"
   "Tag_38" := "DB_Tagforce".Status."Step"."2";
   IF #_w1 THEN "DB_Tagforce".Lock."Step"."2" := TRUE; END_IF;
   #_w2 := "DB_Tagforce".Lock."Step"."2" AND "DB_Tanks".Source.Caustic.Sensor.High AND NOT "Tag_39";   // rising edge of "DB_Tanks".Source.Caustic.Sensor.High
   "Tag_39" := "DB_Tanks".Source.Caustic.Sensor.High;
   IF #_w2 THEN
       "DB_Tanks".Source.Caustic.Valve.Source := FALSE;
       "DB_Tanks".Source.Caustic.Object.Pump := FALSE;
       "DB_Counter".Caustic := TRUE;
   END_IF;
   #_w3 := "DB_Tagforce".Lock."Step"."2" AND "DB_Tanks".Source.Acid.Sensor.High AND NOT "Tag_40";   // rising edge of "DB_Tanks".Source.Acid.Sensor.High
   "Tag_40" := "DB_Tanks".Source.Acid.Sensor.High;
   IF #_w3 THEN
       "DB_Tanks".Source.Acid.Valve.Source := FALSE;
       "DB_Tanks".Source.Acid.Object.Pump := FALSE;
       "DB_Counter".Acid := TRUE;
   END_IF;
   #_w4 := "DB_Tagforce".Lock."Step"."2" AND "DB_Tanks".Source.Water.Sensor.High AND NOT "Tag_41";   // rising edge of "DB_Tanks".Source.Water.Sensor.High
   "Tag_41" := "DB_Tanks".Source.Water.Sensor.High;
   IF #_w4 THEN
       "DB_Tanks".Source.Water.Valve.Source := FALSE;
       "DB_Tanks".Source.Water.Object.Pump := FALSE;
       "DB_Counter".Water := TRUE;
   END_IF;
   IF "DB_Tagforce".Lock."Step"."2" AND NOT "DB_Tanks".Source.Caustic.Sensor.High THEN
       "DB_Tanks".Source.Caustic.Valve.Source := TRUE;
       "DB_Tanks".Source.Caustic.Object.Pump := TRUE;
   END_IF;
   IF "DB_Tagforce".Lock."Step"."2" AND NOT "DB_Tanks".Source.Acid.Sensor.High THEN
       "DB_Tanks".Source.Acid.Valve.Source := TRUE;
       "DB_Tanks".Source.Acid.Object.Pump := TRUE;
   END_IF;
   IF "DB_Tagforce".Lock."Step"."2" AND NOT "DB_Tanks".Source.Water.Sensor.High THEN
       "DB_Tanks".Source.Water.Valve.Source := TRUE;
       "DB_Tanks".Source.Water.Object.Pump := TRUE;
   END_IF;
   IF "DB_Tagforce".Lock."Step"."2" AND "DB_Tanks".Source.Caustic.Sensor.High AND "DB_Tanks".Source.Acid.Sensor.High AND "DB_Tanks".Source.Water.Sensor.High THEN
       "DB_Tagforce".Lock."Step"."2" := FALSE;
   END_IF;
   "IEC_Timer_0_DB_20".TON(IN := "DB_Tagforce".Status."Step"."2" AND "DB_Tanks".Source.Caustic.Sensor.High AND "DB_Tanks".Source.Acid.Sensor.High AND "DB_Tanks".Source.Water.Sensor.High,
                           PT := T#2s);
   IF "IEC_Timer_0_DB_20".Q THEN "DB_Tagforce".Status."Step"."2" := FALSE; END_IF;
   #_w5 := NOT "DB_Tagforce".Status."Step"."2" AND "Tag_59";   // falling edge of "DB_Tagforce".Status."Step"."2"
   "Tag_59" := "DB_Tagforce".Status."Step"."2";
   IF #_w5 AND "DB_Tagforce".Status.Program.Offline THEN "DB_Tagforce".Status."Step"."2" := FALSE; END_IF;
END_REGION

REGION Network 7: Step 3: Pre Rinse
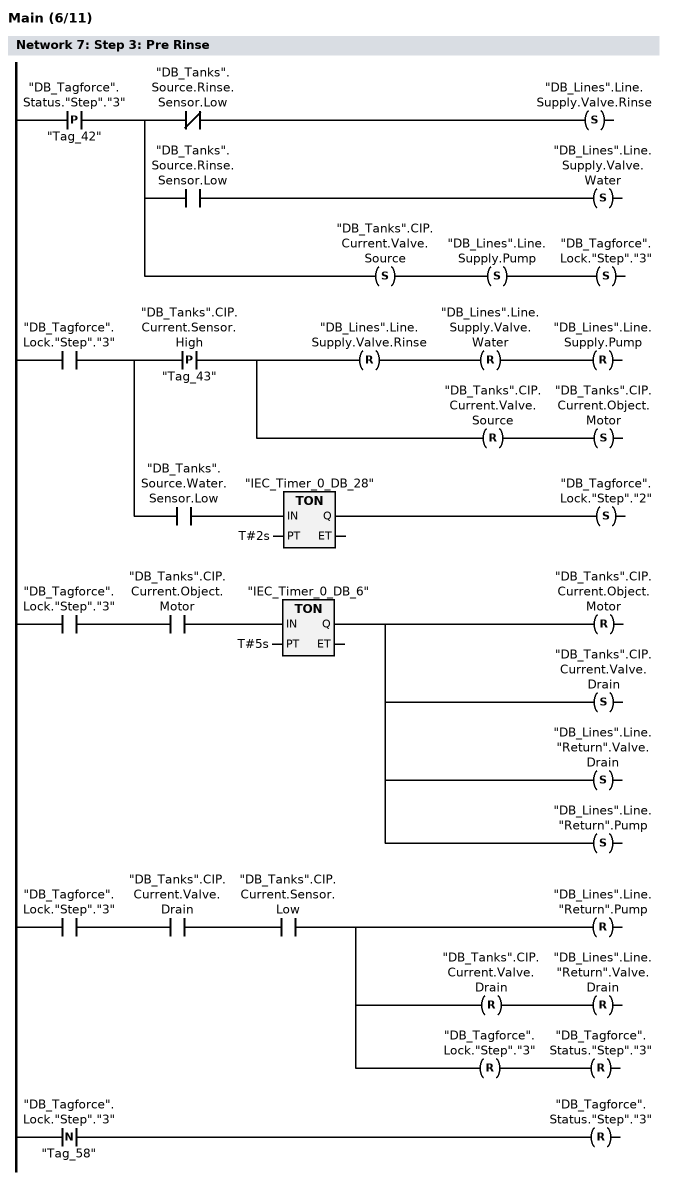
   #_w1 := "DB_Tagforce".Status."Step"."3" AND NOT "Tag_42";   // rising edge of "DB_Tagforce".Status."Step"."3"
   "Tag_42" := "DB_Tagforce".Status."Step"."3";
   IF #_w1 AND NOT "DB_Tanks".Source.Rinse.Sensor.Low THEN
       "DB_Lines".Line.Supply.Valve.Rinse := TRUE;
   END_IF;
   IF #_w1 AND "DB_Tanks".Source.Rinse.Sensor.Low THEN "DB_Lines".Line.Supply.Valve.Water := TRUE; END_IF;
   IF #_w1 THEN
       "DB_Tanks".CIP.Current.Valve.Source := TRUE;
       "DB_Lines".Line.Supply.Pump := TRUE;
       "DB_Tagforce".Lock."Step"."3" := TRUE;
   END_IF;
   #_w2 := "DB_Tagforce".Lock."Step"."3" AND "DB_Tanks".CIP.Current.Sensor.High AND NOT "Tag_43";   // rising edge of "DB_Tanks".CIP.Current.Sensor.High
   "Tag_43" := "DB_Tanks".CIP.Current.Sensor.High;
   IF #_w2 THEN
       "DB_Lines".Line.Supply.Valve.Rinse := FALSE;
       "DB_Lines".Line.Supply.Valve.Water := FALSE;
       "DB_Lines".Line.Supply.Pump := FALSE;
       "DB_Tanks".CIP.Current.Valve.Source := FALSE;
       "DB_Tanks".CIP.Current.Object.Motor := TRUE;
   END_IF;
   "IEC_Timer_0_DB_28".TON(IN := "DB_Tagforce".Lock."Step"."3" AND "DB_Tanks".Source.Water.Sensor.Low,
                           PT := T#2s);
   IF "IEC_Timer_0_DB_28".Q THEN "DB_Tagforce".Lock."Step"."2" := TRUE; END_IF;
   "IEC_Timer_0_DB_6".TON(IN := "DB_Tagforce".Lock."Step"."3" AND "DB_Tanks".CIP.Current.Object.Motor,
                          PT := T#5s);
   IF "IEC_Timer_0_DB_6".Q THEN
       "DB_Tanks".CIP.Current.Object.Motor := FALSE;
       "DB_Tanks".CIP.Current.Valve.Drain := TRUE;
       "DB_Lines".Line."Return".Valve.Drain := TRUE;
       "DB_Lines".Line."Return".Pump := TRUE;
   END_IF;
   IF "DB_Tagforce".Lock."Step"."3" AND "DB_Tanks".CIP.Current.Valve.Drain AND "DB_Tanks".CIP.Current.Sensor.Low THEN
       "DB_Lines".Line."Return".Pump := FALSE;
   END_IF;
   #_w3 := "DB_Tagforce".Lock."Step"."3" AND "DB_Tanks".CIP.Current.Valve.Drain AND "DB_Tanks".CIP.Current.Sensor.Low;
   IF #_w3 THEN
       "DB_Tanks".CIP.Current.Valve.Drain := FALSE;
       "DB_Lines".Line."Return".Valve.Drain := FALSE;
       "DB_Tagforce".Lock."Step"."3" := FALSE;
       "DB_Tagforce".Status."Step"."3" := FALSE;
   END_IF;
   #_w4 := NOT "DB_Tagforce".Lock."Step"."3" AND "Tag_58";   // falling edge of "DB_Tagforce".Lock."Step"."3"
   "Tag_58" := "DB_Tagforce".Lock."Step"."3";
   IF #_w4 THEN "DB_Tagforce".Status."Step"."3" := FALSE; END_IF;
END_REGION

REGION Network 8: Step 4: Caustic Wash
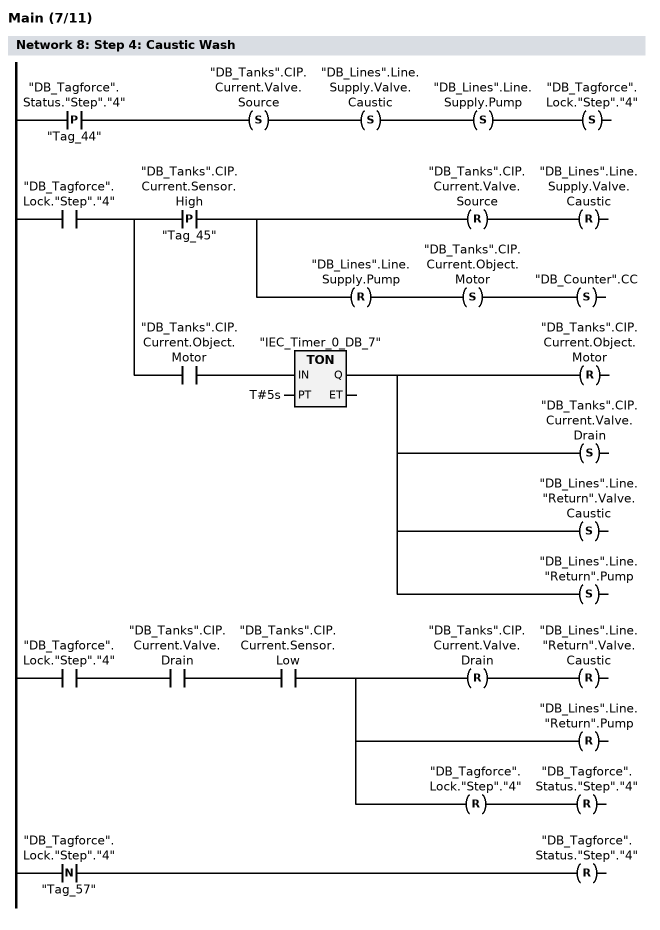
   #_w1 := "DB_Tagforce".Status."Step"."4" AND NOT "Tag_44";   // rising edge of "DB_Tagforce".Status."Step"."4"
   "Tag_44" := "DB_Tagforce".Status."Step"."4";
   IF #_w1 THEN
       "DB_Tanks".CIP.Current.Valve.Source := TRUE;
       "DB_Lines".Line.Supply.Valve.Caustic := TRUE;
       "DB_Lines".Line.Supply.Pump := TRUE;
       "DB_Tagforce".Lock."Step"."4" := TRUE;
   END_IF;
   #_w2 := "DB_Tagforce".Lock."Step"."4" AND "DB_Tanks".CIP.Current.Sensor.High AND NOT "Tag_45";   // rising edge of "DB_Tanks".CIP.Current.Sensor.High
   "Tag_45" := "DB_Tanks".CIP.Current.Sensor.High;
   IF #_w2 THEN
       "DB_Tanks".CIP.Current.Valve.Source := FALSE;
       "DB_Lines".Line.Supply.Valve.Caustic := FALSE;
       "DB_Lines".Line.Supply.Pump := FALSE;
       "DB_Tanks".CIP.Current.Object.Motor := TRUE;
       "DB_Counter".CC := TRUE;
   END_IF;
   "IEC_Timer_0_DB_7".TON(IN := "DB_Tagforce".Lock."Step"."4" AND "DB_Tanks".CIP.Current.Object.Motor,
                          PT := T#5s);
   IF "IEC_Timer_0_DB_7".Q THEN
       "DB_Tanks".CIP.Current.Object.Motor := FALSE;
       "DB_Tanks".CIP.Current.Valve.Drain := TRUE;
       "DB_Lines".Line."Return".Valve.Caustic := TRUE;
       "DB_Lines".Line."Return".Pump := TRUE;
   END_IF;
   #_w3 := "DB_Tagforce".Lock."Step"."4" AND "DB_Tanks".CIP.Current.Valve.Drain AND "DB_Tanks".CIP.Current.Sensor.Low;
   IF #_w3 THEN
       "DB_Tanks".CIP.Current.Valve.Drain := FALSE;
       "DB_Lines".Line."Return".Valve.Caustic := FALSE;
       "DB_Lines".Line."Return".Pump := FALSE;
       "DB_Tagforce".Lock."Step"."4" := FALSE;
       "DB_Tagforce".Status."Step"."4" := FALSE;
   END_IF;
   #_w4 := NOT "DB_Tagforce".Lock."Step"."4" AND "Tag_57";   // falling edge of "DB_Tagforce".Lock."Step"."4"
   "Tag_57" := "DB_Tagforce".Lock."Step"."4";
   IF #_w4 THEN "DB_Tagforce".Status."Step"."4" := FALSE; END_IF;
END_REGION

REGION Network 9: Step 5: Intermediate Rinse
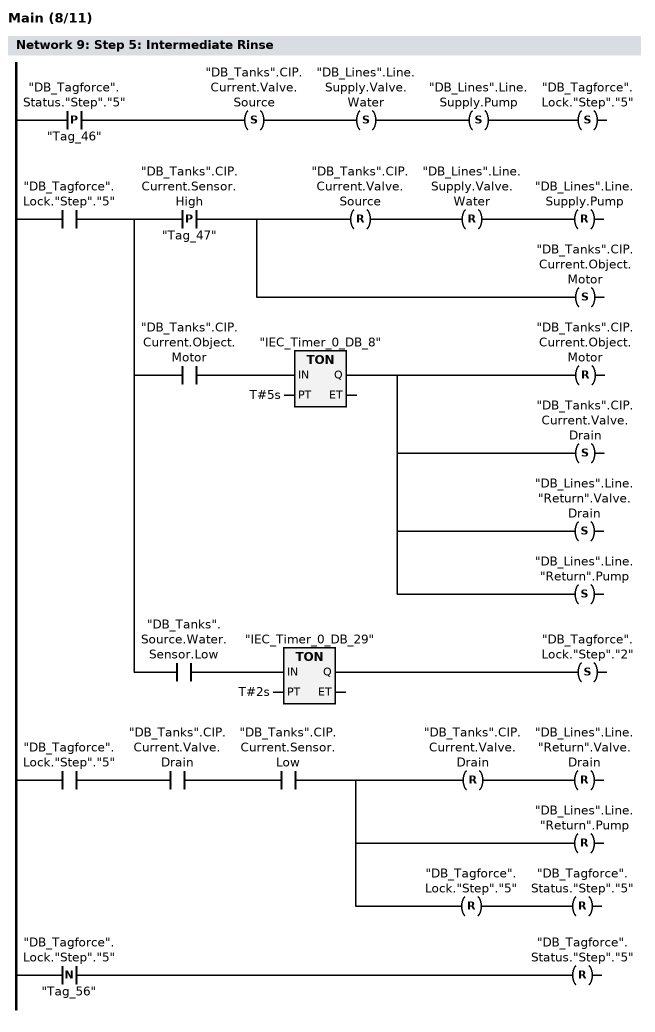
   #_w1 := "DB_Tagforce".Status."Step"."5" AND NOT "Tag_46";   // rising edge of "DB_Tagforce".Status."Step"."5"
   "Tag_46" := "DB_Tagforce".Status."Step"."5";
   IF #_w1 THEN
       "DB_Tanks".CIP.Current.Valve.Source := TRUE;
       "DB_Lines".Line.Supply.Valve.Water := TRUE;
       "DB_Lines".Line.Supply.Pump := TRUE;
       "DB_Tagforce".Lock."Step"."5" := TRUE;
   END_IF;
   #_w2 := "DB_Tagforce".Lock."Step"."5" AND "DB_Tanks".CIP.Current.Sensor.High AND NOT "Tag_47";   // rising edge of "DB_Tanks".CIP.Current.Sensor.High
   "Tag_47" := "DB_Tanks".CIP.Current.Sensor.High;
   IF #_w2 THEN
       "DB_Tanks".CIP.Current.Valve.Source := FALSE;
       "DB_Lines".Line.Supply.Valve.Water := FALSE;
       "DB_Lines".Line.Supply.Pump := FALSE;
       "DB_Tanks".CIP.Current.Object.Motor := TRUE;
   END_IF;
   "IEC_Timer_0_DB_8".TON(IN := "DB_Tagforce".Lock."Step"."5" AND "DB_Tanks".CIP.Current.Object.Motor,
                          PT := T#5s);
   IF "IEC_Timer_0_DB_8".Q THEN
       "DB_Tanks".CIP.Current.Object.Motor := FALSE;
       "DB_Tanks".CIP.Current.Valve.Drain := TRUE;
       "DB_Lines".Line."Return".Valve.Drain := TRUE;
       "DB_Lines".Line."Return".Pump := TRUE;
   END_IF;
   "IEC_Timer_0_DB_29".TON(IN := "DB_Tagforce".Lock."Step"."5" AND "DB_Tanks".Source.Water.Sensor.Low,
                           PT := T#2s);
   IF "IEC_Timer_0_DB_29".Q THEN "DB_Tagforce".Lock."Step"."2" := TRUE; END_IF;
   #_w3 := "DB_Tagforce".Lock."Step"."5" AND "DB_Tanks".CIP.Current.Valve.Drain AND "DB_Tanks".CIP.Current.Sensor.Low;
   IF #_w3 THEN
       "DB_Tanks".CIP.Current.Valve.Drain := FALSE;
       "DB_Lines".Line."Return".Valve.Drain := FALSE;
       "DB_Lines".Line."Return".Pump := FALSE;
       "DB_Tagforce".Lock."Step"."5" := FALSE;
       "DB_Tagforce".Status."Step"."5" := FALSE;
   END_IF;
   #_w4 := NOT "DB_Tagforce".Lock."Step"."5" AND "Tag_56";   // falling edge of "DB_Tagforce".Lock."Step"."5"
   "Tag_56" := "DB_Tagforce".Lock."Step"."5";
   IF #_w4 THEN "DB_Tagforce".Status."Step"."5" := FALSE; END_IF;
END_REGION

REGION Network 10: Step 6: Acid Wash
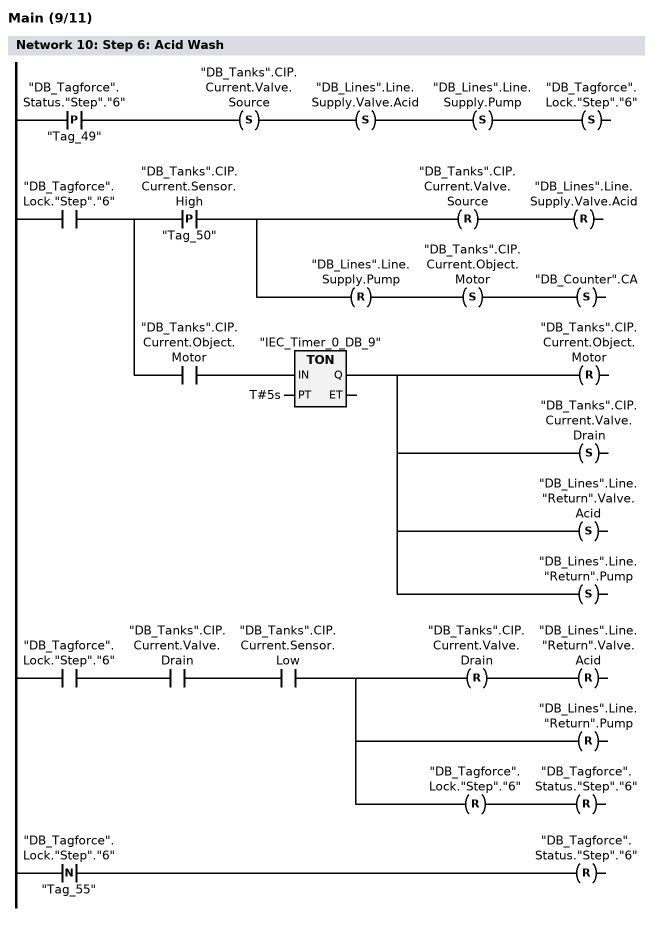
   #_w1 := "DB_Tagforce".Status."Step"."6" AND NOT "Tag_49";   // rising edge of "DB_Tagforce".Status."Step"."6"
   "Tag_49" := "DB_Tagforce".Status."Step"."6";
   IF #_w1 THEN
       "DB_Tanks".CIP.Current.Valve.Source := TRUE;
       "DB_Lines".Line.Supply.Valve.Acid := TRUE;
       "DB_Lines".Line.Supply.Pump := TRUE;
       "DB_Tagforce".Lock."Step"."6" := TRUE;
   END_IF;
   #_w2 := "DB_Tagforce".Lock."Step"."6" AND "DB_Tanks".CIP.Current.Sensor.High AND NOT "Tag_50";   // rising edge of "DB_Tanks".CIP.Current.Sensor.High
   "Tag_50" := "DB_Tanks".CIP.Current.Sensor.High;
   IF #_w2 THEN
       "DB_Tanks".CIP.Current.Valve.Source := FALSE;
       "DB_Lines".Line.Supply.Valve.Acid := FALSE;
       "DB_Lines".Line.Supply.Pump := FALSE;
       "DB_Tanks".CIP.Current.Object.Motor := TRUE;
       "DB_Counter".CA := TRUE;
   END_IF;
   "IEC_Timer_0_DB_9".TON(IN := "DB_Tagforce".Lock."Step"."6" AND "DB_Tanks".CIP.Current.Object.Motor,
                          PT := T#5s);
   IF "IEC_Timer_0_DB_9".Q THEN
       "DB_Tanks".CIP.Current.Object.Motor := FALSE;
       "DB_Tanks".CIP.Current.Valve.Drain := TRUE;
       "DB_Lines".Line."Return".Valve.Acid := TRUE;
       "DB_Lines".Line."Return".Pump := TRUE;
   END_IF;
   #_w3 := "DB_Tagforce".Lock."Step"."6" AND "DB_Tanks".CIP.Current.Valve.Drain AND "DB_Tanks".CIP.Current.Sensor.Low;
   IF #_w3 THEN
       "DB_Tanks".CIP.Current.Valve.Drain := FALSE;
       "DB_Lines".Line."Return".Valve.Acid := FALSE;
       "DB_Lines".Line."Return".Pump := FALSE;
       "DB_Tagforce".Lock."Step"."6" := FALSE;
       "DB_Tagforce".Status."Step"."6" := FALSE;
   END_IF;
   #_w4 := NOT "DB_Tagforce".Lock."Step"."6" AND "Tag_55";   // falling edge of "DB_Tagforce".Lock."Step"."6"
   "Tag_55" := "DB_Tagforce".Lock."Step"."6";
   IF #_w4 THEN "DB_Tagforce".Status."Step"."6" := FALSE; END_IF;
END_REGION

REGION Network 11: Step 7: Final Rinse
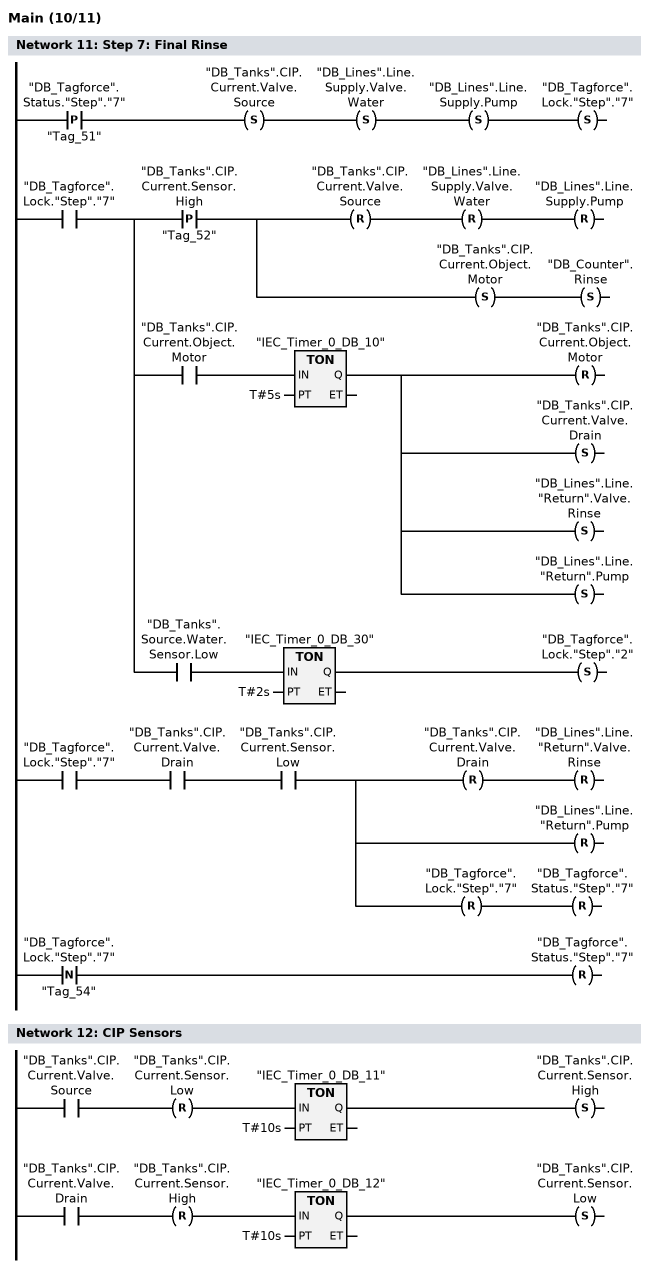
   #_w1 := "DB_Tagforce".Status."Step"."7" AND NOT "Tag_51";   // rising edge of "DB_Tagforce".Status."Step"."7"
   "Tag_51" := "DB_Tagforce".Status."Step"."7";
   IF #_w1 THEN
       "DB_Tanks".CIP.Current.Valve.Source := TRUE;
       "DB_Lines".Line.Supply.Valve.Water := TRUE;
       "DB_Lines".Line.Supply.Pump := TRUE;
       "DB_Tagforce".Lock."Step"."7" := TRUE;
   END_IF;
   #_w2 := "DB_Tagforce".Lock."Step"."7" AND "DB_Tanks".CIP.Current.Sensor.High AND NOT "Tag_52";   // rising edge of "DB_Tanks".CIP.Current.Sensor.High
   "Tag_52" := "DB_Tanks".CIP.Current.Sensor.High;
   IF #_w2 THEN
       "DB_Tanks".CIP.Current.Valve.Source := FALSE;
       "DB_Lines".Line.Supply.Valve.Water := FALSE;
       "DB_Lines".Line.Supply.Pump := FALSE;
       "DB_Tanks".CIP.Current.Object.Motor := TRUE;
       "DB_Counter".Rinse := TRUE;
   END_IF;
   "IEC_Timer_0_DB_10".TON(IN := "DB_Tagforce".Lock."Step"."7" AND "DB_Tanks".CIP.Current.Object.Motor,
                           PT := T#5s);
   IF "IEC_Timer_0_DB_10".Q THEN
       "DB_Tanks".CIP.Current.Object.Motor := FALSE;
       "DB_Tanks".CIP.Current.Valve.Drain := TRUE;
       "DB_Lines".Line."Return".Valve.Rinse := TRUE;
       "DB_Lines".Line."Return".Pump := TRUE;
   END_IF;
   "IEC_Timer_0_DB_30".TON(IN := "DB_Tagforce".Lock."Step"."7" AND "DB_Tanks".Source.Water.Sensor.Low,
                           PT := T#2s);
   IF "IEC_Timer_0_DB_30".Q THEN "DB_Tagforce".Lock."Step"."2" := TRUE; END_IF;
   #_w3 := "DB_Tagforce".Lock."Step"."7" AND "DB_Tanks".CIP.Current.Valve.Drain AND "DB_Tanks".CIP.Current.Sensor.Low;
   IF #_w3 THEN
       "DB_Tanks".CIP.Current.Valve.Drain := FALSE;
       "DB_Lines".Line."Return".Valve.Rinse := FALSE;
       "DB_Lines".Line."Return".Pump := FALSE;
       "DB_Tagforce".Lock."Step"."7" := FALSE;
       "DB_Tagforce".Status."Step"."7" := FALSE;
   END_IF;
   #_w4 := NOT "DB_Tagforce".Lock."Step"."7" AND "Tag_54";   // falling edge of "DB_Tagforce".Lock."Step"."7"
   "Tag_54" := "DB_Tagforce".Lock."Step"."7";
   IF #_w4 THEN "DB_Tagforce".Status."Step"."7" := FALSE; END_IF;
END_REGION

REGION Network 12: CIP Sensors
   IF "DB_Tanks".CIP.Current.Valve.Source THEN "DB_Tanks".CIP.Current.Sensor.Low := FALSE; END_IF;
   "IEC_Timer_0_DB_11".TON(IN := "DB_Tanks".CIP.Current.Valve.Source, PT := T#10s);
   IF "IEC_Timer_0_DB_11".Q THEN "DB_Tanks".CIP.Current.Sensor.High := TRUE; END_IF;
   IF "DB_Tanks".CIP.Current.Valve.Drain THEN "DB_Tanks".CIP.Current.Sensor.High := FALSE; END_IF;
   "IEC_Timer_0_DB_12".TON(IN := "DB_Tanks".CIP.Current.Valve.Drain, PT := T#10s);
   IF "IEC_Timer_0_DB_12".Q THEN "DB_Tanks".CIP.Current.Sensor.Low := TRUE; END_IF;
END_REGION

REGION Network 13: Sources
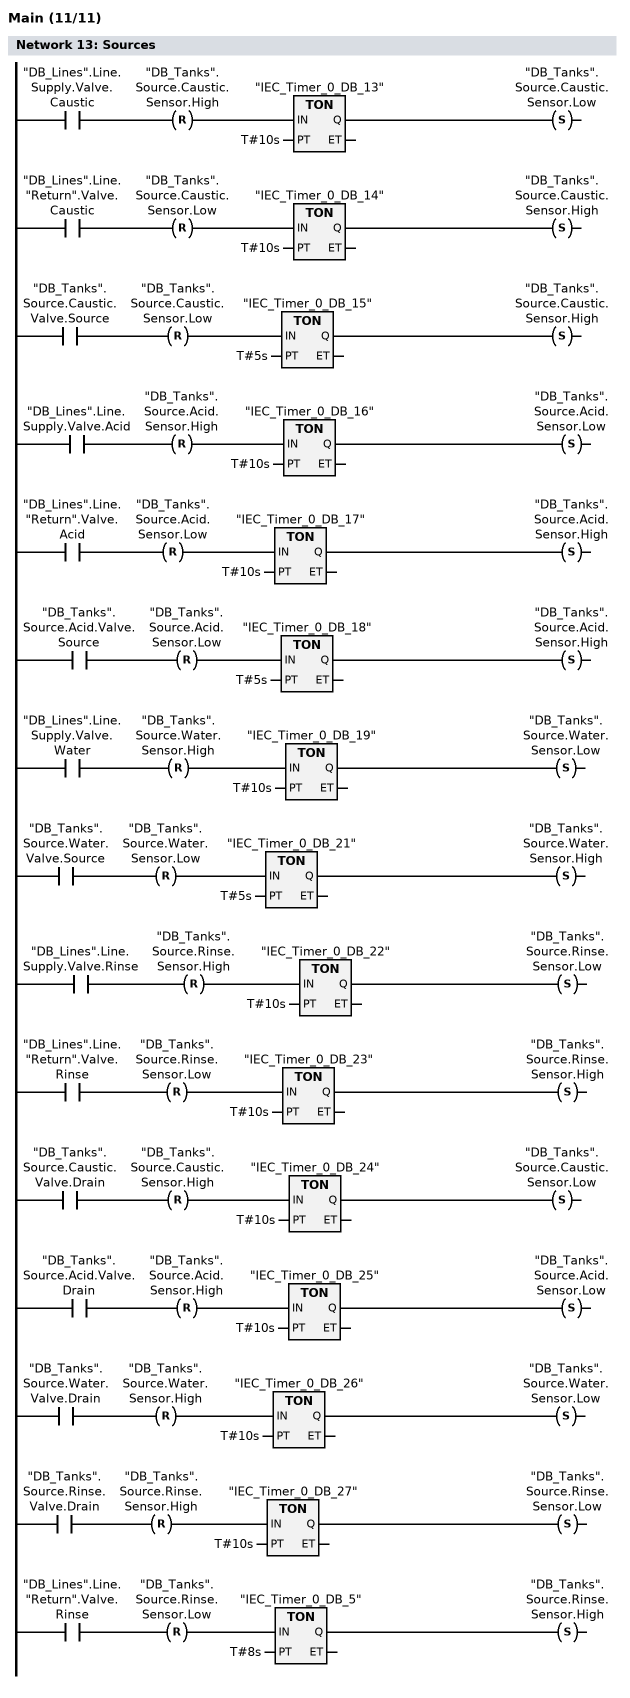
   IF "DB_Lines".Line.Supply.Valve.Caustic THEN "DB_Tanks".Source.Caustic.Sensor.High := FALSE; END_IF;
   "IEC_Timer_0_DB_13".TON(IN := "DB_Lines".Line.Supply.Valve.Caustic, PT := T#10s);
   IF "IEC_Timer_0_DB_13".Q THEN "DB_Tanks".Source.Caustic.Sensor.Low := TRUE; END_IF;
   IF "DB_Lines".Line."Return".Valve.Caustic THEN "DB_Tanks".Source.Caustic.Sensor.Low := FALSE; END_IF;
   "IEC_Timer_0_DB_14".TON(IN := "DB_Lines".Line."Return".Valve.Caustic, PT := T#10s);
   IF "IEC_Timer_0_DB_14".Q THEN "DB_Tanks".Source.Caustic.Sensor.High := TRUE; END_IF;
   IF "DB_Tanks".Source.Caustic.Valve.Source THEN "DB_Tanks".Source.Caustic.Sensor.Low := FALSE; END_IF;
   "IEC_Timer_0_DB_15".TON(IN := "DB_Tanks".Source.Caustic.Valve.Source, PT := T#5s);
   IF "IEC_Timer_0_DB_15".Q THEN "DB_Tanks".Source.Caustic.Sensor.High := TRUE; END_IF;
   IF "DB_Lines".Line.Supply.Valve.Acid THEN "DB_Tanks".Source.Acid.Sensor.High := FALSE; END_IF;
   "IEC_Timer_0_DB_16".TON(IN := "DB_Lines".Line.Supply.Valve.Acid, PT := T#10s);
   IF "IEC_Timer_0_DB_16".Q THEN "DB_Tanks".Source.Acid.Sensor.Low := TRUE; END_IF;
   IF "DB_Lines".Line."Return".Valve.Acid THEN "DB_Tanks".Source.Acid.Sensor.Low := FALSE; END_IF;
   "IEC_Timer_0_DB_17".TON(IN := "DB_Lines".Line."Return".Valve.Acid, PT := T#10s);
   IF "IEC_Timer_0_DB_17".Q THEN "DB_Tanks".Source.Acid.Sensor.High := TRUE; END_IF;
   IF "DB_Tanks".Source.Acid.Valve.Source THEN "DB_Tanks".Source.Acid.Sensor.Low := FALSE; END_IF;
   "IEC_Timer_0_DB_18".TON(IN := "DB_Tanks".Source.Acid.Valve.Source, PT := T#5s);
   IF "IEC_Timer_0_DB_18".Q THEN "DB_Tanks".Source.Acid.Sensor.High := TRUE; END_IF;
   IF "DB_Lines".Line.Supply.Valve.Water THEN "DB_Tanks".Source.Water.Sensor.High := FALSE; END_IF;
   "IEC_Timer_0_DB_19".TON(IN := "DB_Lines".Line.Supply.Valve.Water, PT := T#10s);
   IF "IEC_Timer_0_DB_19".Q THEN "DB_Tanks".Source.Water.Sensor.Low := TRUE; END_IF;
   IF "DB_Tanks".Source.Water.Valve.Source THEN "DB_Tanks".Source.Water.Sensor.Low := FALSE; END_IF;
   "IEC_Timer_0_DB_21".TON(IN := "DB_Tanks".Source.Water.Valve.Source, PT := T#5s);
   IF "IEC_Timer_0_DB_21".Q THEN "DB_Tanks".Source.Water.Sensor.High := TRUE; END_IF;
   IF "DB_Lines".Line.Supply.Valve.Rinse THEN "DB_Tanks".Source.Rinse.Sensor.High := FALSE; END_IF;
   "IEC_Timer_0_DB_22".TON(IN := "DB_Lines".Line.Supply.Valve.Rinse, PT := T#10s);
   IF "IEC_Timer_0_DB_22".Q THEN "DB_Tanks".Source.Rinse.Sensor.Low := TRUE; END_IF;
   IF "DB_Lines".Line."Return".Valve.Rinse THEN "DB_Tanks".Source.Rinse.Sensor.Low := FALSE; END_IF;
   "IEC_Timer_0_DB_23".TON(IN := "DB_Lines".Line."Return".Valve.Rinse, PT := T#10s);
   IF "IEC_Timer_0_DB_23".Q THEN "DB_Tanks".Source.Rinse.Sensor.High := TRUE; END_IF;
   IF "DB_Tanks".Source.Caustic.Valve.Drain THEN "DB_Tanks".Source.Caustic.Sensor.High := FALSE; END_IF;
   "IEC_Timer_0_DB_24".TON(IN := "DB_Tanks".Source.Caustic.Valve.Drain, PT := T#10s);
   IF "IEC_Timer_0_DB_24".Q THEN "DB_Tanks".Source.Caustic.Sensor.Low := TRUE; END_IF;
   IF "DB_Tanks".Source.Acid.Valve.Drain THEN "DB_Tanks".Source.Acid.Sensor.High := FALSE; END_IF;
   "IEC_Timer_0_DB_25".TON(IN := "DB_Tanks".Source.Acid.Valve.Drain, PT := T#10s);
   IF "IEC_Timer_0_DB_25".Q THEN "DB_Tanks".Source.Acid.Sensor.Low := TRUE; END_IF;
   IF "DB_Tanks".Source.Water.Valve.Drain THEN "DB_Tanks".Source.Water.Sensor.High := FALSE; END_IF;
   "IEC_Timer_0_DB_26".TON(IN := "DB_Tanks".Source.Water.Valve.Drain, PT := T#10s);
   IF "IEC_Timer_0_DB_26".Q THEN "DB_Tanks".Source.Water.Sensor.Low := TRUE; END_IF;
   IF "DB_Tanks".Source.Rinse.Valve.Drain THEN "DB_Tanks".Source.Rinse.Sensor.High := FALSE; END_IF;
   "IEC_Timer_0_DB_27".TON(IN := "DB_Tanks".Source.Rinse.Valve.Drain, PT := T#10s);
   IF "IEC_Timer_0_DB_27".Q THEN "DB_Tanks".Source.Rinse.Sensor.Low := TRUE; END_IF;
   IF "DB_Lines".Line."Return".Valve.Rinse THEN "DB_Tanks".Source.Rinse.Sensor.Low := FALSE; END_IF;
   "IEC_Timer_0_DB_5".TON(IN := "DB_Lines".Line."Return".Valve.Rinse, PT := T#8s);
   IF "IEC_Timer_0_DB_5".Q THEN "DB_Tanks".Source.Rinse.Sensor.High := TRUE; END_IF;
END_REGION
END_ORGANIZATION_BLOCK